C01819=1031.307,-50.754,414.134,167.850,42.108,157.823
C01820=1031.301,-51.003,414.145,167.848,42.110,157.824
C01821=1031.295,-51.252,414.157,167.845,42.111,157.824
C01822=1031.289,-51.502,414.170,167.842,42.113,157.824
C01823=1031.282,-51.752,414.182,167.840,42.114,157.824
C01824=1031.274,-52.034,414.195,167.836,42.116,157.824
C01825=1031.267,-52.314,414.209,167.834,42.117,157.824
C01826=1031.261,-52.596,414.222,167.831,42.119,157.824
C01827=1031.253,-52.877,414.236,167.827,42.120,157.824
C01828=1031.247,-53.127,414.247,167.824,42.122,157.824
C01829=1031.241,-53.376,414.259,167.822,42.123,157.824
C01830=1031.235,-53.626,414.271,167.820,42.124,157.824
C01831=1031.228,-53.875,414.283,167.817,42.126,157.824
C01832=1031.222,-54.125,414.296,167.814,42.127,157.824
C01833=1031.215,-54.375,414.308,167.811,42.128,157.824
C01834=1031.209,-54.624,414.320,167.809,42.130,157.825
C01835=1031.204,-54.874,414.331,167.806,42.131,157.825
C01836=1031.197,-55.124,414.343,167.803,42.133,157.825
C01837=1031.191,-55.373,414.355,167.800,42.134,157.825
C01838=1031.184,-55.623,414.367,167.797,42.136,157.825
C01839=1031.179,-55.872,414.379,167.795,42.137,157.825
C01840=1031.172,-56.122,414.391,167.792,42.139,157.825
C01841=1031.166,-56.372,414.402,167.789,42.140,157.825
C01842=1031.159,-56.621,414.414,167.786,42.141,157.825
C01843=1031.153,-56.871,414.427,167.783,42.143,157.825
C01844=1031.147,-57.120,414.439,167.782,42.144,157.825
C01845=1031.141,-57.370,414.450,167.779,42.145,157.825
C01846=1031.135,-57.620,414.462,167.776,42.146,157.825
C01847=1031.128,-57.870,414.474,167.773,42.148,157.826
C01848=1031.122,-58.119,414.485,167.771,42.149,157.826
C01849=1031.116,-58.369,414.497,167.768,42.150,157.826
C01850=1031.110,-58.619,414.510,167.765,42.152,157.826
C01851=1031.104,-58.867,414.521,167.762,42.153,157.826
C01852=1031.097,-59.118,414.533,167.759,42.155,157.826
C01853=1031.091,-59.367,414.545,167.757,42.156,157.826
C01854=1031.085,-59.617,414.557,167.754,42.158,157.826
C01855=1031.079,-59.867,414.568,167.751,42.159,157.826
C01856=1031.072,-60.116,414.580,167.748,42.161,157.826
C01857=1031.066,-60.366,414.592,167.745,42.162,157.826
C01858=1031.061,-60.616,414.603,167.743,42.163,157.826
C01859=1031.054,-60.865,414.615,167.740,42.165,157.826
C01860=1031.048,-61.115,414.627,167.737,42.166,157.826
C01861=1031.042,-61.364,414.638,167.735,42.168,157.826
C01862=1031.036,-61.614,414.651,167.732,42.169,157.826
C01863=1031.030,-61.864,414.662,167.730,42.170,157.827
C01864=1031.023,-62.113,414.674,167.727,42.172,157.827
C01865=1031.017,-62.363,414.685,167.724,42.173,157.827
C01866=1031.010,-62.613,414.697,167.721,42.174,157.827
C01867=1031.005,-62.862,414.709,167.718,42.176,157.827
C01868=1030.999,-63.112,414.720,167.716,42.177,157.827
C01869=1030.993,-63.361,414.732,167.713,42.178,157.827
C01870=1030.986,-63.611,414.743,167.710,42.180,157.827
C01871=1030.981,-63.861,414.756,167.707,42.181,157.827
C01872=1030.975,-64.111,414.766,167.704,42.182,157.827
C01873=1030.968,-64.360,414.778,167.702,42.184,157.827
C01874=1030.962,-64.610,414.789,167.699,42.185,157.827
C01875=1030.956,-64.859,414.801,167.696,42.187,157.827
C01876=1030.951,-65.109,414.813,167.693,42.188,157.827
C01877=1030.944,-65.359,414.825,167.690,42.189,157.827
C01878=1030.938,-65.609,414.836,167.688,42.191,157.827
C01879=1030.932,-65.858,414.848,167.685,42.192,157.828
C01880=1030.925,-66.108,414.859,167.683,42.194,157.828
C01881=1030.920,-66.357,414.871,167.680,42.195,157.828
C01882=1030.914,-66.607,414.882,167.678,42.197,157.828
C01883=1030.908,-66.857,414.893,167.675,42.198,157.828
C01884=1030.901,-67.106,414.905,167.672,42.199,157.828
C01885=1030.896,-67.356,414.916,167.669,42.201,157.828
C01886=1030.890,-67.606,414.928,167.666,42.202,157.828
C01887=1030.884,-67.855,414.939,167.664,42.204,157.828
C01888=1030.877,-68.138,414.952,167.660,42.205,157.828
C01889=1030.870,-68.421,414.965,167.657,42.207,157.828
C01890=1030.863,-68.703,414.978,167.654,42.208,157.828
C01891=1030.856,-68.986,414.991,167.651,42.210,157.828
C01892=1030.851,-69.235,415.003,167.648,42.211,157.828
C01893=1030.845,-69.485,415.014,167.646,42.212,157.828
C01894=1030.839,-69.735,415.025,167.643,42.213,157.828
C01895=1030.832,-69.984,415.037,167.640,42.215,157.829
C01896=1030.826,-70.234,415.048,167.638,42.216,157.829
C01897=1030.820,-70.484,415.059,167.635,42.217,157.829
C01898=1030.815,-70.733,415.071,167.632,42.219,157.829
C01899=1030.809,-70.983,415.083,167.629,42.220,157.829
C01900=1030.803,-71.233,415.093,167.626,42.222,157.829
C01901=1030.797,-71.481,415.105,167.624,42.223,157.829
C01902=1030.790,-71.732,415.116,167.621,42.225,157.829
C01903=1030.785,-71.981,415.127,167.618,42.226,157.829
C01904=1030.779,-72.232,415.139,167.615,42.227,157.829
C01905=1030.773,-72.481,415.151,167.612,42.229,157.829
C01906=1030.767,-72.730,415.161,167.610,42.230,157.829
C01907=1030.761,-72.980,415.173,167.607,42.232,157.829
C01908=1030.755,-73.230,415.184,167.604,42.233,157.829
C01909=1030.749,-73.480,415.195,167.601,42.234,157.829
C01910=1030.744,-73.729,415.207,167.598,42.236,157.829
C01911=1030.738,-73.979,415.218,167.596,42.237,157.829
C01912=1030.731,-74.229,415.229,167.593,42.239,157.830
C01913=1030.726,-74.478,415.240,167.590,42.240,157.830
C01914=1030.720,-74.728,415.251,167.587,42.242,157.830
C01915=1030.713,-74.978,415.262,167.584,42.243,157.830
C01916=1030.707,-75.227,415.272,167.582,42.245,157.830
C01917=1030.701,-75.477,415.284,167.579,42.246,157.830
C01918=1030.695,-75.727,415.295,167.576,42.247,157.830
C01919=1030.689,-75.976,415.305,167.574,42.249,157.830
C01920=1030.683,-76.226,415.317,167.571,42.250,157.830
C01921=1030.677,-76.475,415.328,167.568,42.252,157.830
C01922=1030.671,-76.725,415.339,167.565,42.254,157.830
C01923=1030.664,-76.975,415.350,167.562,42.255,157.830
C01924=1030.658,-77.224,415.361,167.560,42.257,157.831
C01925=1030.653,-77.474,415.372,167.557,42.258,157.831
C01926=1030.646,-77.724,415.383,167.554,42.260,157.831
C01927=1030.641,-77.973,415.394,167.551,42.261,157.831
C01928=1030.635,-78.223,415.405,167.549,42.263,157.831
C01929=1030.629,-78.474,415.415,167.546,42.264,157.831
C01930=1030.622,-78.723,415.425,167.543,42.265,157.831
C01931=1030.617,-78.972,415.436,167.540,42.267,157.831
C01932=1030.610,-79.223,415.447,167.538,42.269,157.831
C01933=1030.604,-79.472,415.458,167.534,42.270,157.831
C01934=1030.599,-79.722,415.469,167.531,42.272,157.831
C01935=1030.593,-79.971,415.480,167.528,42.273,157.831
C01936=1030.586,-80.221,415.491,167.525,42.275,157.831
C01937=1030.580,-80.470,415.502,167.523,42.277,157.832
C01938=1030.574,-80.720,415.512,167.520,42.279,157.832
C01939=1030.568,-80.970,415.522,167.517,42.280,157.832
C01940=1030.562,-81.220,415.533,167.515,42.281,157.832
C01941=1030.555,-81.469,415.544,167.512,42.283,157.832
C01942=1030.549,-81.719,415.555,167.509,42.285,157.832
C01943=1030.543,-81.969,415.566,167.506,42.287,157.832
C01944=1030.537,-82.219,415.575,167.503,42.288,157.832
C01945=1030.531,-82.468,415.586,167.500,42.290,157.832
C01946=1030.524,-82.718,415.597,167.497,42.292,157.832
C01947=1030.519,-82.967,415.608,167.495,42.293,157.833
C01948=1030.513,-83.218,415.618,167.492,42.295,157.833
C01949=1030.507,-83.467,415.628,167.489,42.296,157.833
C01950=1030.500,-83.717,415.639,167.486,42.298,157.833
C01951=1030.494,-83.967,415.649,167.484,42.300,157.833
C01952=1030.487,-84.251,415.662,167.480,42.302,157.833
C01953=1030.480,-84.535,415.674,167.477,42.304,157.833
C01954=1030.474,-84.820,415.685,167.474,42.306,157.833
C01955=1030.467,-85.105,415.697,167.471,42.307,157.833
C01956=1030.461,-85.354,415.708,167.468,42.309,157.834
C01957=1030.455,-85.604,415.718,167.464,42.310,157.834
C01958=1030.449,-85.854,415.729,167.462,42.312,157.834
C01959=1030.443,-86.104,415.739,167.459,42.314,157.834
C01960=1030.437,-86.353,415.750,167.456,42.316,157.834
C01961=1030.430,-86.603,415.760,167.453,42.317,157.834
C01962=1030.425,-86.853,415.770,167.451,42.319,157.834
C01963=1030.418,-87.102,415.780,167.448,42.321,157.834
C01964=1030.412,-87.352,415.791,167.445,42.322,157.834
C01965=1030.407,-87.602,415.802,167.442,42.323,157.834
C01966=1030.400,-87.851,415.812,167.439,42.325,157.834
C01967=1030.395,-88.101,415.822,167.436,42.327,157.835
C01968=1030.388,-88.351,415.832,167.433,42.329,157.835
C01969=1030.383,-88.601,415.843,167.431,42.331,157.835
C01970=1030.376,-88.850,415.853,167.428,42.332,157.835
C01971=1030.371,-89.100,415.863,167.425,42.334,157.835
C01972=1030.364,-89.349,415.873,167.422,42.336,157.835
C01973=1030.358,-89.599,415.885,167.420,42.337,157.835
C01974=1030.353,-89.849,415.895,167.417,42.338,157.835
C01975=1030.346,-90.099,415.905,167.413,42.340,157.835
C01976=1030.341,-90.349,415.915,167.410,42.342,157.835
C01977=1030.334,-90.598,415.925,167.408,42.344,157.836
C01978=1030.329,-90.848,415.936,167.405,42.346,157.836
C01979=1030.323,-91.098,415.945,167.402,42.347,157.836
C01980=1030.317,-91.347,415.956,167.399,42.349,157.836
C01981=1030.311,-91.597,415.966,167.397,42.350,157.836
C01982=1030.305,-91.847,415.976,167.394,42.352,157.836
C01983=1030.299,-92.096,415.986,167.391,42.353,157.836
C01984=1030.293,-92.346,415.997,167.388,42.355,157.836
C01985=1030.287,-92.596,416.006,167.385,42.357,157.836
C01986=1030.282,-92.846,416.017,167.382,42.359,157.836
C01987=1030.275,-93.095,416.027,167.379,42.360,157.836
C01988=1030.270,-93.345,416.037,167.377,42.362,157.836
C01989=1030.264,-93.595,416.048,167.374,42.364,157.837
C01990=1030.258,-93.844,416.058,167.371,42.365,157.837
C01991=1030.252,-94.095,416.068,167.369,42.367,157.837
C01992=1030.246,-94.344,416.078,167.366,42.368,157.837
C01993=1030.240,-94.594,416.088,167.362,42.370,157.837
C01994=1030.234,-94.844,416.098,167.359,42.372,157.837
C01995=1030.228,-95.093,416.109,167.357,42.374,157.837
C01996=1030.222,-95.343,416.118,167.354,42.375,157.837
C01997=1030.217,-95.593,416.128,167.351,42.377,157.837
C01998=1030.210,-95.842,416.139,167.348,42.379,157.837
C01999=1030.205,-96.092,416.149,167.346,42.380,157.838
C02000=1030.199,-96.342,416.158,167.343,42.382,157.838
C02001=1030.193,-96.592,416.169,167.340,42.383,157.838
C02002=1030.187,-96.841,416.179,167.336,42.385,157.838
C02003=1030.182,-97.091,416.189,167.334,42.387,157.838
C02004=1030.176,-97.341,416.198,167.331,42.389,157.838
C02005=1030.170,-97.590,416.209,167.328,42.390,157.838
C02006=1030.164,-97.840,416.219,167.325,42.392,157.838
C02007=1030.158,-98.090,416.228,167.323,42.394,157.838
C02008=1030.152,-98.339,416.238,167.320,42.395,157.838
C02009=1030.146,-98.590,416.248,167.316,42.397,157.839
C02010=1030.140,-98.839,416.257,167.314,42.399,157.839
C02011=1030.134,-99.089,416.267,167.311,42.401,157.839
C02012=1030.127,-99.338,416.277,167.308,42.403,157.839
C02013=1030.122,-99.588,416.287,167.306,42.405,157.839
C02014=1030.116,-99.838,416.297,167.302,42.407,157.839
C02015=1030.110,-100.087,416.306,167.299,42.408,157.839
C02016=1030.103,-100.375,416.317,167.297,42.410,157.839
C02017=1030.096,-100.661,416.328,167.293,42.413,157.840
C02018=1030.090,-100.948,416.340,167.289,42.415,157.840
C02019=1030.083,-101.236,416.351,167.287,42.417,157.840
C02020=1030.077,-101.485,416.360,167.284,42.418,157.840
C02021=1030.071,-101.734,416.370,167.280,42.420,157.840
C02022=1030.065,-101.984,416.379,167.278,42.422,157.840
C02023=1030.060,-102.234,416.389,167.275,42.424,157.840
C02024=1030.053,-102.484,416.399,167.272,42.426,157.840
C02025=1030.047,-102.734,416.409,167.269,42.428,157.840
C02026=1030.042,-102.983,416.418,167.266,42.429,157.841
C02027=1030.035,-103.233,416.427,167.263,42.431,157.841
C02028=1030.030,-103.483,416.438,167.260,42.433,157.841
C02029=1030.024,-103.733,416.447,167.258,42.435,157.841
C02030=1030.018,-103.983,416.457,167.255,42.437,157.841
C02031=1030.012,-104.232,416.466,167.252,42.439,157.841
C02032=1030.006,-104.481,416.475,167.249,42.440,157.841
C02033=1030.001,-104.732,416.486,167.246,42.442,157.841
C02034=1029.994,-104.981,416.495,167.243,42.444,157.842
C02035=1029.988,-105.231,416.505,167.241,42.446,157.842
C02036=1029.983,-105.480,416.514,167.238,42.448,157.842
C02037=1029.976,-105.730,416.524,167.234,42.450,157.842
C02038=1029.970,-105.980,416.533,167.231,42.451,157.842
C02039=1029.965,-106.230,416.543,167.229,42.453,157.842
C02040=1029.960,-106.480,416.552,167.226,42.455,157.842
C02041=1029.953,-106.729,416.561,167.223,42.457,157.842
C02042=1029.947,-106.979,416.571,167.220,42.459,157.842
C02043=1029.941,-107.229,416.580,167.217,42.461,157.843
C02044=1029.935,-107.478,416.590,167.214,42.462,157.843
C02045=1029.930,-107.729,416.598,167.212,42.464,157.843
C02046=1029.923,-107.978,416.608,167.209,42.466,157.843
C02047=1029.918,-108.227,416.617,167.205,42.468,157.843
C02048=1029.912,-108.477,416.627,167.203,42.470,157.843
C02049=1029.906,-108.727,416.636,167.200,42.472,157.843
C02050=1029.900,-108.977,416.645,167.197,42.473,157.843
C02051=1029.894,-109.227,416.654,167.195,42.475,157.843
C02052=1029.888,-109.476,416.664,167.191,42.478,157.844
C02053=1029.882,-109.727,416.673,167.188,42.480,157.844
C02054=1029.876,-109.976,416.682,167.186,42.482,157.844
C02055=1029.870,-110.226,416.692,167.183,42.483,157.844
C02056=1029.864,-110.475,416.701,167.179,42.485,157.844
C02057=1029.859,-110.725,416.710,167.177,42.487,157.844
C02058=1029.853,-110.975,416.719,167.174,42.489,157.844
C02059=1029.847,-111.225,416.729,167.171,42.491,157.845
C02060=1029.841,-111.474,416.737,167.168,42.493,157.845
C02061=1029.835,-111.724,416.747,167.165,42.495,157.845
C02062=1029.829,-111.975,416.756,167.162,42.497,157.845
C02063=1029.824,-112.224,416.765,167.160,42.499,157.845
C02064=1029.817,-112.474,416.774,167.157,42.501,157.845
C02065=1029.812,-112.723,416.783,167.153,42.503,157.845
C02066=1029.806,-112.973,416.793,167.151,42.504,157.845
C02067=1029.800,-113.223,416.802,167.148,42.506,157.846
C02068=1029.795,-113.473,416.811,167.145,42.508,157.846
C02069=1029.788,-113.722,416.820,167.143,42.511,157.846
C02070=1029.783,-113.972,416.829,167.139,42.513,157.846
C02071=1029.777,-114.222,416.838,167.136,42.514,157.846
C02072=1029.771,-114.472,416.847,167.134,42.516,157.846
C02073=1029.766,-114.721,416.856,167.131,42.518,157.846
C02074=1029.760,-114.972,416.865,167.127,42.520,157.846
C02075=1029.754,-115.221,416.874,167.125,42.522,157.847
C02076=1029.748,-115.471,416.883,167.122,42.524,157.847
C02077=1029.742,-115.720,416.892,167.119,42.526,157.847
C02078=1029.736,-115.971,416.901,167.116,42.528,157.847
C02079=1029.731,-116.220,416.910,167.113,42.530,157.847
C02080=1029.724,-116.506,416.921,167.109,42.533,157.847
C02081=1029.717,-116.793,416.930,167.107,42.534,157.847
C02082=1029.711,-117.079,416.941,167.103,42.537,157.848
C02083=1029.703,-117.365,416.951,167.100,42.539,157.848
C02084=1029.698,-117.615,416.960,167.097,42.541,157.848
C02085=1029.692,-117.866,416.968,167.094,42.543,157.848
C02086=1029.686,-118.115,416.978,167.091,42.545,157.848
C02087=1029.680,-118.365,416.986,167.088,42.547,157.848
C02088=1029.674,-118.614,416.995,167.085,42.550,157.849
C02089=1029.668,-118.864,417.004,167.083,42.551,157.849
C02090=1029.663,-119.114,417.012,167.079,42.553,157.849
C02091=1029.657,-119.364,417.022,167.076,42.555,157.849
C02092=1029.651,-119.613,417.030,167.074,42.558,157.849
C02093=1029.645,-119.864,417.039,167.071,42.560,157.849
C02094=1029.639,-120.113,417.048,167.067,42.562,157.849
C02095=1029.634,-120.362,417.056,167.065,42.563,157.849
C02096=1029.628,-120.612,417.065,167.062,42.566,157.850
C02097=1029.622,-120.862,417.073,167.060,42.568,157.850
C02098=1029.616,-121.112,417.083,167.056,42.570,157.850
C02099=1029.611,-121.362,417.091,167.053,42.571,157.850
C02100=1029.605,-121.612,417.100,167.051,42.574,157.850
C02101=1029.599,-121.861,417.109,167.048,42.576,157.850
C02102=1029.593,-122.111,417.117,167.044,42.578,157.850
C02103=1029.588,-122.361,417.126,167.042,42.580,157.851
C02104=1029.582,-122.610,417.134,167.039,42.582,157.851
C02105=1029.576,-122.861,417.143,167.036,42.584,157.851
C02106=1029.570,-123.110,417.152,167.033,42.586,157.851
C02107=1029.564,-123.360,417.161,167.030,42.588,157.851
C02108=1029.558,-123.610,417.169,167.028,42.590,157.851
C02109=1029.553,-123.859,417.177,167.025,42.592,157.851
C02110=1029.547,-124.110,417.186,167.021,42.594,157.852
C02111=1029.542,-124.359,417.195,167.019,42.597,157.852
C02112=1029.536,-124.608,417.203,167.016,42.598,157.852
C02113=1029.530,-124.859,417.212,167.012,42.600,157.852
C02114=1029.524,-125.108,417.220,167.010,42.603,157.852
C02115=1029.518,-125.359,417.229,167.007,42.605,157.852
C02116=1029.513,-125.608,417.237,167.004,42.607,157.852
C02117=1029.507,-125.858,417.245,167.001,42.609,157.853
C02118=1029.501,-126.108,417.254,166.998,42.611,157.853
C02119=1029.495,-126.358,417.262,166.996,42.614,157.853
C02120=1029.489,-126.607,417.270,166.992,42.615,157.853
C02121=1029.484,-126.858,417.279,166.989,42.617,157.853
C02122=1029.478,-127.107,417.287,166.987,42.620,157.853
C02123=1029.472,-127.357,417.295,166.984,42.622,157.854
C02124=1029.466,-127.606,417.304,166.980,42.624,157.854
C02125=1029.461,-127.855,417.313,166.978,42.626,157.854
C02126=1029.455,-128.106,417.321,166.975,42.628,157.854
C02127=1029.450,-128.355,417.331,166.972,42.629,157.854
C02128=1029.446,-128.604,417.340,166.970,42.630,157.854
C02129=1029.443,-128.855,417.351,166.968,42.631,157.854
C02130=1029.440,-129.104,417.362,166.964,42.630,157.854
C02131=1029.437,-129.354,417.374,166.962,42.630,157.853
C02132=1029.436,-129.604,417.386,166.960,42.629,157.853
C02133=1029.435,-129.853,417.399,166.958,42.627,157.853
C02134=1029.435,-130.103,417.412,166.955,42.625,157.852
C02135=1029.435,-130.353,417.426,166.954,42.623,157.852
C02136=1029.435,-130.603,417.440,166.952,42.620,157.851
C02137=1029.436,-130.853,417.456,166.950,42.617,157.850
C02138=1029.439,-131.103,417.472,166.948,42.613,157.850
C02139=1029.441,-131.352,417.488,166.947,42.608,157.849
C02140=1029.445,-131.603,417.505,166.945,42.604,157.848
C02141=1029.448,-131.853,417.523,166.944,42.599,157.847
C02142=1029.453,-132.103,417.540,166.942,42.593,157.846
C02143=1029.458,-132.352,417.560,166.941,42.586,157.845
C02144=1029.141,-132.377,417.253,166.892,42.832,157.882
C02145=1029.137,-132.128,417.233,166.894,42.838,157.883
C02146=1029.132,-131.879,417.215,166.895,42.844,157.884
C02147=1029.128,-131.628,417.198,166.896,42.849,157.885
C02148=1029.125,-131.378,417.181,166.898,42.854,157.886
C02149=1029.122,-131.128,417.165,166.900,42.858,157.887
C02150=1029.120,-130.878,417.149,166.902,42.862,157.888
C02151=1029.119,-130.628,417.133,166.903,42.865,157.889
C02152=1029.118,-130.378,417.119,166.905,42.868,157.889
C02153=1029.118,-130.128,417.105,166.907,42.871,157.890
C02154=1029.118,-129.878,417.092,166.909,42.872,157.890
C02155=1029.119,-129.629,417.078,166.911,42.874,157.891
C02156=1029.121,-129.379,417.066,166.914,42.875,157.891
C02157=1029.123,-129.129,417.054,166.916,42.876,157.891
C02158=1029.126,-128.880,417.044,166.918,42.876,157.891
C02159=1029.129,-128.630,417.033,166.921,42.876,157.892
C02160=1029.134,-128.381,417.023,166.923,42.875,157.892
C02161=1029.138,-128.131,417.014,166.926,42.873,157.892
C02162=1029.143,-127.880,417.005,166.929,42.872,157.891
C02163=1029.150,-127.631,416.996,166.932,42.869,157.891
C02164=1029.155,-127.382,416.988,166.935,42.867,157.891
C02165=1029.161,-127.132,416.980,166.937,42.865,157.891
C02166=1029.166,-126.882,416.971,166.941,42.863,157.891
C02167=1029.173,-126.632,416.963,166.944,42.861,157.891
C02168=1029.178,-126.383,416.955,166.946,42.858,157.891
C02169=1029.184,-126.133,416.947,166.950,42.856,157.890
C02170=1029.190,-125.883,416.938,166.953,42.854,157.890
C02171=1029.195,-125.633,416.929,166.955,42.852,157.890
C02172=1029.201,-125.384,416.921,166.959,42.850,157.890
C02173=1029.207,-125.133,416.913,166.961,42.847,157.890
C02174=1029.213,-124.884,416.905,166.964,42.845,157.890
C02175=1029.218,-124.634,416.896,166.968,42.843,157.889
C02176=1029.224,-124.384,416.887,166.970,42.841,157.889
C02177=1029.230,-124.135,416.879,166.973,42.839,157.889
C02178=1029.236,-123.885,416.870,166.975,42.836,157.889
C02179=1029.242,-123.635,416.861,166.979,42.834,157.889
C02180=1029.247,-123.385,416.853,166.982,42.833,157.889
C02181=1029.253,-123.136,416.845,166.984,42.830,157.889
C02182=1029.259,-122.886,416.835,166.988,42.828,157.888
C02183=1029.264,-122.636,416.827,166.991,42.826,157.888
C02184=1029.271,-122.386,416.819,166.993,42.824,157.888
C02185=1029.276,-122.136,416.810,166.996,42.822,157.888
C02186=1029.281,-121.887,416.802,166.999,42.820,157.888
C02187=1029.288,-121.637,416.792,167.002,42.817,157.888
C02188=1029.294,-121.387,416.784,167.005,42.816,157.888
C02189=1029.299,-121.137,416.775,167.008,42.814,157.888
C02190=1029.305,-120.887,416.767,167.011,42.811,157.887
C02191=1029.311,-120.638,416.757,167.013,42.809,157.887
C02192=1029.317,-120.388,416.750,167.016,42.807,157.887
C02193=1029.322,-120.138,416.741,167.020,42.805,157.887
C02194=1029.328,-119.889,416.731,167.022,42.803,157.887
C02195=1029.334,-119.639,416.723,167.025,42.801,157.887
C02196=1029.339,-119.388,416.714,167.029,42.799,157.887
C02197=1029.345,-119.139,416.706,167.031,42.796,157.886
C02198=1029.352,-118.889,416.697,167.034,42.795,157.886
C02199=1029.357,-118.640,416.688,167.037,42.793,157.886
C02200=1029.363,-118.390,416.679,167.040,42.791,157.886
C02201=1029.369,-118.140,416.671,167.043,42.788,157.886
C02202=1029.375,-117.890,416.662,167.045,42.786,157.886
C02203=1029.380,-117.641,416.653,167.049,42.784,157.886
C02204=1029.386,-117.390,416.644,167.052,42.782,157.885
C02205=1029.393,-117.105,416.634,167.055,42.780,157.885
C02206=1029.400,-116.818,416.624,167.058,42.777,157.885
C02207=1029.406,-116.532,416.614,167.061,42.775,157.885
C02208=1029.413,-116.245,416.603,167.065,42.773,157.885
C02209=1029.418,-115.996,416.595,167.068,42.771,157.885
C02210=1029.425,-115.746,416.585,167.070,42.769,157.885
C02211=1029.430,-115.496,416.576,167.074,42.766,157.884
C02212=1029.437,-115.247,416.567,167.077,42.764,157.884
C02213=1029.442,-114.997,416.559,167.079,42.763,157.884
C02214=1029.448,-114.747,416.549,167.082,42.761,157.884
C02215=1029.454,-114.497,416.541,167.085,42.758,157.884
C02216=1029.460,-114.248,416.531,167.088,42.756,157.884
C02217=1029.465,-113.997,416.523,167.091,42.754,157.884
C02218=1029.471,-113.748,416.513,167.093,42.753,157.883
C02219=1029.477,-113.498,416.504,167.097,42.751,157.883
C02220=1029.482,-113.249,416.495,167.100,42.748,157.883
C02221=1029.488,-112.998,416.486,167.102,42.746,157.883
C02222=1029.495,-112.748,416.477,167.105,42.744,157.883
C02223=1029.500,-112.499,416.468,167.109,42.742,157.883
C02224=1029.506,-112.249,416.459,167.111,42.741,157.883
C02225=1029.512,-112.000,416.450,167.114,42.739,157.883
C02226=1029.517,-111.749,416.441,167.117,42.737,157.882
C02227=1029.524,-111.500,416.431,167.120,42.734,157.882
C02228=1029.529,-111.251,416.422,167.123,42.732,157.882
C02229=1029.535,-111.000,416.413,167.126,42.731,157.882
C02230=1029.541,-110.750,416.404,167.128,42.729,157.882
C02231=1029.547,-110.501,416.394,167.132,42.727,157.882
C02232=1029.553,-110.251,416.386,167.135,42.725,157.882
C02233=1029.559,-110.001,416.376,167.137,42.722,157.881
C02234=1029.564,-109.752,416.367,167.140,42.721,157.881
C02235=1029.570,-109.501,416.358,167.143,42.719,157.881
C02236=1029.576,-109.252,416.348,167.146,42.717,157.881
C02237=1029.582,-109.003,416.339,167.149,42.715,157.881
C02238=1029.588,-108.753,416.330,167.151,42.713,157.881
C02239=1029.594,-108.502,416.321,167.155,42.711,157.881
C02240=1029.600,-108.253,416.312,167.158,42.709,157.881
C02241=1029.606,-108.003,416.302,167.160,42.707,157.880
C02242=1029.612,-107.754,416.292,167.163,42.705,157.880
C02243=1029.618,-107.503,416.284,167.167,42.703,157.880
C02244=1029.623,-107.254,416.274,167.169,42.701,157.880
C02245=1029.630,-107.004,416.265,167.172,42.699,157.880
C02246=1029.636,-106.755,416.255,167.175,42.698,157.880
C02247=1029.641,-106.505,416.246,167.178,42.696,157.880
C02248=1029.647,-106.255,416.237,167.181,42.693,157.880
C02249=1029.653,-106.005,416.228,167.184,42.691,157.879
C02250=1029.659,-105.755,416.217,167.186,42.689,157.879
C02251=1029.664,-105.506,416.208,167.189,42.688,157.879
C02252=1029.670,-105.256,416.199,167.193,42.686,157.879
C02253=1029.677,-105.006,416.189,167.195,42.684,157.879
C02254=1029.683,-104.757,416.180,167.198,42.682,157.879
C02255=1029.688,-104.508,416.170,167.201,42.680,157.879
C02256=1029.694,-104.257,416.161,167.204,42.678,157.879
C02257=1029.700,-104.007,416.151,167.207,42.676,157.879
C02258=1029.706,-103.757,416.142,167.210,42.674,157.878
C02259=1029.711,-103.508,416.133,167.212,42.673,157.878
C02260=1029.718,-103.258,416.123,167.215,42.671,157.878
C02261=1029.723,-103.008,416.113,167.219,42.669,157.878
C02262=1029.729,-102.758,416.103,167.222,42.667,157.878
C02263=1029.735,-102.509,416.094,167.224,42.665,157.878
C02264=1029.741,-102.260,416.084,167.227,42.663,157.878
C02265=1029.746,-102.009,416.074,167.230,42.662,157.878
C02266=1029.753,-101.760,416.065,167.233,42.660,157.878
C02267=1029.759,-101.510,416.055,167.236,42.658,157.877
C02268=1029.765,-101.260,416.046,167.239,42.656,157.877
C02269=1029.772,-100.973,416.035,167.242,42.653,157.877
C02270=1029.778,-100.687,416.024,167.245,42.651,157.877
C02271=1029.785,-100.400,416.011,167.248,42.649,157.877
C02272=1029.792,-100.113,416.000,167.252,42.647,157.877
C02273=1029.798,-99.863,415.991,167.255,42.646,157.877
C02274=1029.804,-99.614,415.981,167.257,42.643,157.876
C02275=1029.810,-99.365,415.972,167.260,42.641,157.876
C02276=1029.815,-99.114,415.962,167.264,42.639,157.876
C02277=1029.821,-98.865,415.952,167.266,42.638,157.876
C02278=1029.828,-98.615,415.943,167.269,42.636,157.876
C02279=1029.834,-98.365,415.933,167.272,42.634,157.876
C02280=1029.839,-98.116,415.922,167.274,42.632,157.876
C02281=1029.846,-97.866,415.913,167.278,42.630,157.876
C02282=1029.852,-97.616,415.903,167.281,42.628,157.876
C02283=1029.857,-97.366,415.893,167.284,42.627,157.876
C02284=1029.863,-97.116,415.884,167.286,42.625,157.875
C02285=1029.869,-96.866,415.873,167.289,42.623,157.875
C02286=1029.875,-96.617,415.863,167.292,42.622,157.875
C02287=1029.880,-96.367,415.853,167.295,42.620,157.875
C02288=1029.886,-96.118,415.844,167.298,42.618,157.875
C02289=1029.892,-95.868,415.833,167.301,42.617,157.875
C02290=1029.898,-95.618,415.823,167.304,42.615,157.875
C02291=1029.904,-95.368,415.813,167.306,42.613,157.875
C02292=1029.910,-95.118,415.804,167.309,42.611,157.875
C02293=1029.916,-94.869,415.793,167.312,42.609,157.875
C02294=1029.922,-94.619,415.783,167.315,42.607,157.874
C02295=1029.927,-94.369,415.773,167.318,42.606,157.874
C02296=1029.934,-94.120,415.763,167.321,42.605,157.874
C02297=1029.939,-93.870,415.752,167.324,42.603,157.874
C02298=1029.945,-93.620,415.743,167.326,42.601,157.874
C02299=1029.951,-93.370,415.732,167.329,42.599,157.874
C02300=1029.957,-93.121,415.722,167.332,42.597,157.874
C02301=1029.963,-92.871,415.712,167.336,42.596,157.874
C02302=1029.969,-92.621,415.702,167.338,42.594,157.874
C02303=1029.975,-92.371,415.692,167.341,42.592,157.874
C02304=1029.981,-92.122,415.682,167.344,42.591,157.873
C02305=1029.986,-91.872,415.671,167.346,42.589,157.873
C02306=1029.993,-91.623,415.661,167.349,42.587,157.873
C02307=1029.998,-91.373,415.651,167.352,42.586,157.873
C02308=1030.005,-91.123,415.641,167.354,42.584,157.873
C02309=1030.010,-90.873,415.631,167.358,42.582,157.873
C02310=1030.016,-90.623,415.620,167.361,42.580,157.873
C02311=1030.022,-90.374,415.610,167.364,42.578,157.873
C02312=1030.028,-90.124,415.600,167.366,42.577,157.873
C02313=1030.034,-89.875,415.590,167.369,42.575,157.873
C02314=1030.040,-89.625,415.579,167.372,42.574,157.873
C02315=1030.046,-89.375,415.569,167.374,42.572,157.872
C02316=1030.051,-89.125,415.559,167.378,42.570,157.872
C02317=1030.058,-88.876,415.549,167.381,42.568,157.872
C02318=1030.064,-88.625,415.538,167.384,42.566,157.872
C02319=1030.070,-88.376,415.528,167.386,42.565,157.872
C02320=1030.076,-88.127,415.517,167.389,42.563,157.872
C02321=1030.082,-87.877,415.507,167.392,42.561,157.872
C02322=1030.088,-87.627,415.497,167.394,42.560,157.872
C02323=1030.094,-87.377,415.486,167.398,42.558,157.872
C02324=1030.100,-87.128,415.476,167.401,42.556,157.872
C02325=1030.105,-86.878,415.466,167.404,42.555,157.872
C02326=1030.113,-86.628,415.455,167.406,42.553,157.871
C02327=1030.118,-86.379,415.444,167.409,42.551,157.871
C02328=1030.124,-86.129,415.434,167.412,42.549,157.871
C02329=1030.130,-85.879,415.424,167.414,42.547,157.871
C02330=1030.136,-85.629,415.414,167.418,42.545,157.871
C02331=1030.142,-85.380,415.404,167.421,42.544,157.871
C02332=1030.148,-85.130,415.392,167.424,42.543,157.871
C02333=1030.155,-84.845,415.380,167.426,42.541,157.871
C02334=1030.163,-84.561,415.369,167.430,42.539,157.871
C02335=1030.169,-84.276,415.357,167.433,42.537,157.870
C02336=1030.176,-83.992,415.345,167.436,42.534,157.870
C02337=1030.182,-83.742,415.334,167.439,42.533,157.870
C02338=1030.188,-83.493,415.324,167.442,42.531,157.870
C02339=1030.194,-83.243,415.314,167.444,42.530,157.870
C02340=1030.201,-82.993,415.303,167.448,42.528,157.870
C02341=1030.207,-82.743,415.292,167.451,42.526,157.870
C02342=1030.212,-82.493,415.282,167.454,42.524,157.870
C02343=1030.218,-82.244,415.272,167.456,42.523,157.870
C02344=1030.225,-81.994,415.261,167.459,42.521,157.870
C02345=1030.231,-81.745,415.250,167.462,42.519,157.869
C02346=1030.237,-81.495,415.240,167.464,42.517,157.869
C02347=1030.242,-81.245,415.229,167.468,42.515,157.869
C02348=1030.250,-80.995,415.219,167.471,42.514,157.869
C02349=1030.255,-80.746,415.208,167.474,42.513,157.869
C02350=1030.261,-80.496,415.197,167.476,42.511,157.869
C02351=1030.268,-80.246,415.187,167.479,42.509,157.869
C02352=1030.274,-79.996,415.176,167.482,42.507,157.869
C02353=1030.279,-79.747,415.165,167.484,42.505,157.869
C02354=1030.286,-79.498,415.155,167.487,42.504,157.869
C02355=1030.292,-79.247,415.144,167.490,42.502,157.868
C02356=1030.298,-78.998,415.133,167.493,42.501,157.868
C02357=1030.304,-78.749,415.122,167.495,42.499,157.868
C02358=1030.310,-78.498,415.111,167.499,42.497,157.868
C02359=1030.316,-78.249,415.100,167.502,42.496,157.868
C02360=1030.321,-77.999,415.089,167.505,42.495,157.868
C02361=1030.328,-77.749,415.078,167.507,42.493,157.868
C02362=1030.334,-77.499,415.068,167.510,42.491,157.868
C02363=1030.340,-77.250,415.057,167.513,42.490,157.868
C02364=1030.345,-77.000,415.046,167.516,42.488,157.868
C02365=1030.352,-76.750,415.035,167.518,42.486,157.868
C02366=1030.357,-76.501,415.024,167.521,42.485,157.868
C02367=1030.364,-76.250,415.013,167.524,42.483,157.867
C02368=1030.370,-76.002,415.001,167.527,42.481,157.867
C02369=1030.376,-75.752,414.991,167.529,42.480,157.867
C02370=1030.383,-75.502,414.980,167.532,42.479,157.867
C02371=1030.388,-75.253,414.969,167.535,42.477,157.867
C02372=1030.394,-75.003,414.958,167.538,42.476,157.867
C02373=1030.400,-74.753,414.947,167.541,42.474,157.867
C02374=1030.406,-74.504,414.936,167.544,42.473,157.867
C02375=1030.412,-74.254,414.925,167.547,42.471,157.867
C02376=1030.418,-74.004,414.914,167.550,42.469,157.867
C02377=1030.424,-73.754,414.903,167.552,42.468,157.867
C02378=1030.430,-73.504,414.892,167.555,42.466,157.867
C02379=1030.436,-73.255,414.880,167.558,42.465,157.867
C02380=1030.442,-73.006,414.869,167.561,42.463,157.866
C02381=1030.448,-72.755,414.858,167.564,42.462,157.866
C02382=1030.453,-72.506,414.847,167.566,42.460,157.866
C02383=1030.459,-72.256,414.836,167.569,42.459,157.866
C02384=1030.466,-72.007,414.824,167.572,42.458,157.866
C02385=1030.472,-71.757,414.813,167.575,42.456,157.866
C02386=1030.478,-71.507,414.802,167.578,42.455,157.866
C02387=1030.484,-71.258,414.791,167.580,42.453,157.866
C02388=1030.489,-71.008,414.779,167.583,42.452,157.866
C02389=1030.495,-70.758,414.767,167.586,42.450,157.866
C02390=1030.501,-70.509,414.756,167.589,42.449,157.866
C02391=1030.508,-70.259,414.745,167.591,42.447,157.866
C02392=1030.513,-70.010,414.734,167.594,42.446,157.866
C02393=1030.519,-69.759,414.722,167.597,42.444,157.866
C02394=1030.525,-69.510,414.711,167.600,42.443,157.866
C02395=1030.531,-69.260,414.699,167.602,42.441,157.866
C02396=1030.537,-69.011,414.688,167.604,42.440,157.866
C02397=1030.544,-68.728,414.675,167.608,42.439,157.865
C02398=1030.551,-68.445,414.662,167.611,42.437,157.865
C02399=1030.557,-68.164,414.649,167.614,42.435,157.865
C02400=1030.565,-67.882,414.636,167.617,42.434,157.865
C02401=1030.570,-67.631,414.625,167.620,42.433,157.865
C02402=1030.576,-67.382,414.614,167.623,42.431,157.865
C02403=1030.583,-67.132,414.602,167.626,42.430,157.865
C02404=1030.588,-66.883,414.591,167.628,42.428,157.865
C02405=1030.595,-66.633,414.579,167.631,42.427,157.865
C02406=1030.600,-66.383,414.567,167.634,42.425,157.865
C02407=1030.607,-66.134,414.555,167.637,42.424,157.865
C02408=1030.612,-65.884,414.545,167.639,42.422,157.865
C02409=1030.619,-65.634,414.533,167.642,42.421,157.865
C02410=1030.625,-65.385,414.522,167.645,42.419,157.865
C02411=1030.630,-65.135,414.510,167.648,42.418,157.865
C02412=1030.637,-64.885,414.498,167.650,42.416,157.864
C02413=1030.643,-64.636,414.487,167.653,42.415,157.864
C02414=1030.649,-64.386,414.475,167.656,42.413,157.864
C02415=1030.655,-64.136,414.464,167.659,42.412,157.864
C02416=1030.661,-63.887,414.452,167.662,42.410,157.864
C02417=1030.667,-63.637,414.441,167.664,42.409,157.864
C02418=1030.673,-63.387,414.429,167.667,42.407,157.864
C02419=1030.680,-63.137,414.418,167.670,42.406,157.864
C02420=1030.685,-62.888,414.405,167.673,42.405,157.864
C02421=1030.691,-62.638,414.394,167.676,42.403,157.864
C02422=1030.698,-62.388,414.382,167.678,42.402,157.864
C02423=1030.704,-62.139,414.371,167.681,42.400,157.864
C02424=1030.710,-61.889,414.359,167.684,42.399,157.864
C02425=1030.716,-61.640,414.347,167.687,42.398,157.864
C02426=1030.722,-61.390,414.336,167.688,42.396,157.863
C02427=1030.729,-61.140,414.324,167.691,42.395,157.863
C02428=1030.734,-60.891,414.313,167.694,42.393,157.863
C02429=1030.740,-60.641,414.301,167.697,42.392,157.863
C02430=1030.747,-60.391,414.289,167.699,42.390,157.863
C02431=1030.753,-60.142,414.278,167.702,42.389,157.863
C02432=1030.759,-59.892,414.266,167.705,42.387,157.863
C02433=1030.765,-59.642,414.253,167.708,42.386,157.863
C02434=1030.771,-59.393,414.242,167.711,42.384,157.863
C02435=1030.778,-59.143,414.230,167.713,42.383,157.863
C02436=1030.784,-58.894,414.218,167.716,42.381,157.863
C02437=1030.790,-58.643,414.207,167.719,42.380,157.863
C02438=1030.796,-58.394,414.195,167.722,42.378,157.863
C02439=1030.803,-58.145,414.183,167.724,42.377,157.863
C02440=1030.809,-57.895,414.172,167.727,42.376,157.862
C02441=1030.814,-57.646,414.160,167.730,42.374,157.862
C02442=1030.821,-57.396,414.148,167.733,42.373,157.862
C02443=1030.828,-57.146,414.136,167.736,42.372,157.862
C02444=1030.834,-56.896,414.124,167.738,42.370,157.862
C02445=1030.839,-56.647,414.112,167.741,42.369,157.862
C02446=1030.846,-56.397,414.100,167.744,42.367,157.862
C02447=1030.853,-56.148,414.088,167.747,42.366,157.862
C02448=1030.859,-55.898,414.077,167.749,42.364,157.862
C02449=1030.864,-55.648,414.065,167.752,42.363,157.862
C02450=1030.871,-55.399,414.053,167.755,42.361,157.862
C02451=1030.877,-55.149,414.041,167.758,42.360,157.862
C02452=1030.883,-54.899,414.029,167.760,42.358,157.862
C02453=1030.890,-54.649,414.017,167.763,42.357,157.862
C02454=1030.896,-54.400,414.006,167.766,42.355,157.861
C02455=1030.902,-54.151,413.994,167.769,42.354,157.861
C02456=1030.908,-53.901,413.981,167.771,42.352,157.861
C02457=1030.915,-53.651,413.969,167.773,42.351,157.861
C02458=1030.921,-53.401,413.958,167.776,42.350,157.861
C02459=1030.927,-53.151,413.945,167.779,42.348,157.861
C02460=1030.933,-52.902,413.934,167.782,42.347,157.861
C02461=1030.941,-52.621,413.920,167.785,42.345,157.861
C02462=1030.948,-52.340,413.906,167.788,42.344,157.861
C02463=1030.955,-52.059,413.892,167.791,42.342,157.861
C02464=1030.962,-51.778,413.879,167.795,42.340,157.861
C02465=1030.969,-51.528,413.867,167.797,42.339,157.861
C02466=1030.974,-51.279,413.855,167.800,42.337,157.861
C02467=1030.981,-51.029,413.843,167.802,42.335,157.860
C02468=1030.988,-50.780,413.831,167.805,42.334,157.860
C02469=1030.994,-50.530,413.819,167.808,42.333,157.860
C02470=1031.000,-50.280,413.807,167.810,42.331,157.860
C02471=1031.006,-50.030,413.794,167.813,42.330,157.860
C02472=1031.012,-49.780,413.782,167.816,42.329,157.860
C02473=1031.018,-49.531,413.769,167.819,42.327,157.860
C02474=1031.024,-49.282,413.757,167.821,42.326,157.860
C02475=1031.030,-49.032,413.745,167.824,42.325,157.860
C02476=1031.036,-48.782,413.732,167.826,42.324,157.860
C02477=1031.042,-48.532,413.720,167.829,42.322,157.860
C02478=1031.048,-48.282,413.708,167.832,42.321,157.860
C02479=1031.055,-48.033,413.696,167.835,42.320,157.860
C02480=1031.061,-47.784,413.683,167.837,42.318,157.860
C02481=1031.067,-47.534,413.670,167.840,42.317,157.860
C02482=1031.073,-47.284,413.658,167.843,42.316,157.860
C02483=1031.079,-47.035,413.646,167.845,42.315,157.860
C02484=1031.085,-46.785,413.633,167.848,42.313,157.860
C02485=1031.091,-46.535,413.621,167.850,42.312,157.860
C02486=1031.098,-46.286,413.608,167.853,42.311,157.860
C02487=1031.104,-46.036,413.596,167.856,42.309,157.859
C02488=1031.110,-45.786,413.583,167.859,42.308,157.859
C02489=1031.116,-45.537,413.571,167.862,42.307,157.859
C02490=1031.122,-45.287,413.559,167.863,42.305,157.859
C02491=1031.128,-45.038,413.545,167.866,42.304,157.859
C02492=1031.135,-44.788,413.533,167.869,42.303,157.859
C02493=1031.141,-44.538,413.521,167.872,42.302,157.859
C02494=1031.147,-44.288,413.508,167.875,42.300,157.859
C02495=1031.154,-44.039,413.496,167.878,42.299,157.859
C02496=1031.160,-43.790,413.483,167.880,42.298,157.859
C02497=1031.166,-43.540,413.470,167.882,42.296,157.859
C02498=1031.172,-43.290,413.458,167.885,42.295,157.859
C02499=1031.178,-43.041,413.445,167.888,42.294,157.859
C02500=1031.184,-42.791,413.433,167.890,42.292,157.859
C02501=1031.190,-42.541,413.420,167.893,42.291,157.859
C02502=1031.197,-42.292,413.407,167.896,42.290,157.859
C02503=1031.203,-42.042,413.395,167.898,42.289,157.859
C02504=1031.209,-41.792,413.382,167.901,42.288,157.859
C02505=1031.216,-41.543,413.370,167.904,42.286,157.859
C02506=1031.222,-41.294,413.357,167.906,42.285,157.858
C02507=1031.228,-41.044,413.345,167.909,42.284,157.858
C02508=1031.234,-40.794,413.331,167.912,42.282,157.858
C02509=1031.241,-40.545,413.319,167.915,42.281,157.858
C02510=1031.247,-40.296,413.306,167.917,42.280,157.858
C02511=1031.253,-40.046,413.293,167.919,42.279,157.858
C02512=1031.259,-39.796,413.281,167.922,42.277,157.858
C02513=1031.266,-39.547,413.268,167.925,42.276,157.858
C02514=1031.272,-39.297,413.256,167.928,42.275,157.858
C02515=1031.278,-39.048,413.242,167.931,42.273,157.858
C02516=1031.284,-38.798,413.230,167.932,42.272,157.858
C02517=1031.290,-38.548,413.217,167.935,42.271,157.858
C02518=1031.297,-38.299,413.205,167.938,42.270,157.858
C02519=1031.303,-38.049,413.191,167.941,42.268,157.858
C02520=1031.309,-37.799,413.178,167.944,42.267,157.858
C02521=1031.315,-37.550,413.165,167.946,42.266,157.858
C02522=1031.321,-37.300,413.153,167.948,42.265,157.858
C02523=1031.328,-37.051,413.139,167.951,42.264,157.858
C02524=1031.334,-36.801,413.127,167.954,42.262,157.858
C02525=1031.341,-36.521,413.112,167.957,42.261,157.858
C02526=1031.347,-36.239,413.097,167.960,42.260,157.857
C02527=1031.354,-35.959,413.082,167.963,42.258,157.857
C02528=1031.361,-35.678,413.068,167.965,42.257,157.857
C02529=1031.367,-35.429,413.055,167.968,42.256,157.857
C02530=1031.373,-35.179,413.042,167.971,42.254,157.857
C02531=1031.380,-34.929,413.029,167.974,42.253,157.857
C02532=1031.386,-34.680,413.015,167.976,42.252,157.857
C02533=1031.392,-34.430,413.003,167.979,42.251,157.857
C02534=1031.398,-34.181,412.990,167.981,42.250,157.857
C02535=1031.404,-33.931,412.977,167.984,42.248,157.857
C02536=1031.410,-33.682,412.964,167.986,42.247,157.857
C02537=1031.417,-33.432,412.950,167.989,42.246,157.857
C02538=1031.423,-33.182,412.938,167.992,42.245,157.857
C02539=1031.429,-32.932,412.924,167.995,42.244,157.857
C02540=1031.436,-32.683,412.911,167.996,42.242,157.857
C02541=1031.442,-32.434,412.898,167.999,42.241,157.857
C02542=1031.448,-32.184,412.885,168.002,42.240,157.857
C02543=1031.455,-31.934,412.872,168.005,42.239,157.857
C02544=1031.461,-31.685,412.858,168.008,42.238,157.857
C02545=1031.467,-31.435,412.846,168.009,42.236,157.857
C02546=1031.473,-31.186,412.832,168.012,42.235,157.857
C02547=1031.479,-30.936,412.819,168.015,42.234,157.857
C02548=1031.486,-30.686,412.806,168.018,42.233,157.857
C02549=1031.492,-30.437,412.793,168.020,42.232,157.857
C02550=1031.498,-30.187,412.780,168.022,42.230,157.856
C02551=1031.504,-29.938,412.766,168.025,42.229,157.856
C02552=1031.511,-29.688,412.753,168.028,42.228,157.856
C02553=1031.517,-29.439,412.740,168.030,42.227,157.856
C02554=1031.523,-29.189,412.727,168.033,42.225,157.856
C02555=1031.529,-28.940,412.714,168.036,42.224,157.856
C02556=1031.536,-28.690,412.700,168.038,42.223,157.856
C02557=1031.542,-28.440,412.687,168.040,42.222,157.856
C02558=1031.549,-28.191,412.674,168.043,42.221,157.856
C02559=1031.555,-27.942,412.660,168.046,42.219,157.856
C02560=1031.561,-27.691,412.647,168.049,42.218,157.856
C02561=1031.568,-27.442,412.634,168.052,42.217,157.856
C02562=1031.574,-27.193,412.621,168.053,42.216,157.856
C02563=1031.580,-26.942,412.607,168.056,42.215,157.856
C02564=1031.586,-26.693,412.593,168.059,42.214,157.856
C02565=1031.592,-26.444,412.580,168.061,42.212,157.856
C02566=1031.598,-26.195,412.567,168.064,42.211,157.856
C02567=1031.605,-25.944,412.553,168.067,42.210,157.856
C02568=1031.611,-25.695,412.539,168.069,42.209,157.856
C02569=1031.617,-25.446,412.526,168.071,42.208,157.856
C02570=1031.623,-25.196,412.512,168.074,42.207,157.856
C02571=1031.629,-24.946,412.499,168.077,42.206,157.856
C02572=1031.635,-24.697,412.485,168.079,42.205,157.856
C02573=1031.642,-24.448,412.472,168.082,42.204,157.856
C02574=1031.648,-24.198,412.458,168.085,42.203,157.855
C02575=1031.654,-23.948,412.445,168.086,42.202,157.855
C02576=1031.660,-23.699,412.431,168.089,42.201,157.855
C02577=1031.666,-23.449,412.417,168.092,42.200,157.855
C02578=1031.673,-23.199,412.404,168.094,42.199,157.855
C02579=1031.679,-22.950,412.390,168.097,42.197,157.855
C02580=1031.685,-22.700,412.376,168.100,42.196,157.855
C02581=1031.691,-22.451,412.363,168.102,42.195,157.855
C02582=1031.697,-22.201,412.350,168.104,42.194,157.855
C02583=1031.704,-21.952,412.335,168.107,42.193,157.855
C02584=1031.710,-21.702,412.321,168.110,42.192,157.855
C02585=1031.717,-21.453,412.308,168.112,42.191,157.855
C02586=1031.723,-21.203,412.295,168.115,42.189,157.855
C02587=1031.728,-20.954,412.281,168.118,42.188,157.855
C02588=1031.735,-20.704,412.267,168.119,42.187,157.855
C02589=1031.742,-20.423,412.251,168.122,42.186,157.855
C02590=1031.749,-20.141,412.236,168.125,42.185,157.855
C02591=1031.756,-19.859,412.220,168.128,42.183,157.855
C02592=1031.764,-19.578,412.205,168.132,42.182,157.855
C02593=1031.769,-19.329,412.191,168.133,42.181,157.855
C02594=1031.776,-19.079,412.178,168.136,42.179,157.855
C02595=1031.782,-18.829,412.164,168.139,42.178,157.855
C02596=1031.788,-18.579,412.150,168.141,42.177,157.855
C02597=1031.795,-18.330,412.137,168.144,42.176,157.855
C02598=1031.802,-18.081,412.122,168.147,42.175,157.855
C02599=1031.807,-17.831,412.109,168.149,42.174,157.855
C02600=1031.813,-17.582,412.095,168.151,42.173,157.855
C02601=1031.820,-17.332,412.082,168.154,42.172,157.855
C02602=1031.826,-17.083,412.067,168.156,42.170,157.854
C02603=1031.833,-16.833,412.053,168.159,42.169,157.854
C02604=1031.839,-16.584,412.040,168.162,42.168,157.854
C02605=1031.845,-16.333,412.026,168.164,42.167,157.854
C02606=1031.852,-16.085,412.012,168.166,42.166,157.854
C02607=1031.859,-15.835,411.998,168.169,42.165,157.854
C02608=1031.864,-15.585,411.984,168.171,42.164,157.854
C02609=1031.871,-15.336,411.970,168.174,42.163,157.854
C02610=1031.877,-15.086,411.956,168.177,42.162,157.854
C02611=1031.883,-14.836,411.943,168.179,42.161,157.854
C02612=1031.889,-14.587,411.928,168.182,42.160,157.854
C02613=1031.895,-14.337,411.914,168.185,42.159,157.854
C02614=1031.902,-14.088,411.900,168.186,42.158,157.854
C02615=1031.908,-13.838,411.886,168.189,42.157,157.854
C02616=1031.914,-13.589,411.872,168.191,42.156,157.854
C02617=1031.920,-13.339,411.857,168.194,42.155,157.854
C02618=1031.926,-13.090,411.844,168.197,42.154,157.854
C02619=1031.933,-12.840,411.829,168.199,42.153,157.854
C02620=1031.939,-12.591,411.815,168.202,42.152,157.854
C02621=1031.946,-12.341,411.801,168.204,42.150,157.854
C02622=1031.951,-12.092,411.787,168.206,42.149,157.854
C02623=1031.958,-11.842,411.772,168.209,42.148,157.854
C02624=1031.964,-11.593,411.759,168.211,42.147,157.854
C02625=1031.970,-11.343,411.744,168.214,42.146,157.854
C02626=1031.977,-11.093,411.730,168.217,42.145,157.854
C02627=1031.983,-10.844,411.716,168.219,42.144,157.854
C02628=1031.989,-10.594,411.701,168.221,42.143,157.854
C02629=1031.995,-10.345,411.687,168.223,42.142,157.854
C02630=1032.001,-10.095,411.673,168.226,42.141,157.854
C02631=1032.008,-9.846,411.659,168.229,42.140,157.854
C02632=1032.014,-9.596,411.645,168.231,42.139,157.854
C02633=1032.020,-9.347,411.630,168.234,42.138,157.854
C02634=1032.027,-9.097,411.617,168.237,42.137,157.853
C02635=1032.033,-8.848,411.602,168.238,42.136,157.853
C02636=1032.039,-8.599,411.588,168.241,42.135,157.853
C02637=1032.046,-8.349,411.574,168.243,42.133,157.853
C02638=1032.051,-8.100,411.559,168.246,42.132,157.853
C02639=1032.058,-7.850,411.545,168.249,42.131,157.853
C02640=1032.065,-7.600,411.531,168.251,42.130,157.853
C02641=1032.070,-7.351,411.516,168.253,42.129,157.853
C02642=1032.077,-7.101,411.502,168.255,42.128,157.853
C02643=1032.084,-6.851,411.487,168.258,42.127,157.853
C02644=1032.090,-6.603,411.473,168.261,42.126,157.853
C02645=1032.096,-6.353,411.459,168.263,42.125,157.853
C02646=1032.103,-6.103,411.444,168.266,42.124,157.853
C02647=1032.109,-5.854,411.430,168.268,42.123,157.853
C02648=1032.115,-5.604,411.416,168.270,42.122,157.853
C02649=1032.121,-5.354,411.401,168.273,42.121,157.853
C02650=1032.128,-5.106,411.387,168.275,42.120,157.853
C02651=1032.134,-4.855,411.373,168.278,42.119,157.853
C02652=1032.140,-4.606,411.358,168.280,42.118,157.853
C02653=1032.148,-4.323,411.342,168.283,42.117,157.853
C02654=1032.155,-4.040,411.325,168.285,42.115,157.853
C02655=1032.162,-3.757,411.309,168.288,42.114,157.853
C02656=1032.169,-3.473,411.293,168.291,42.113,157.853
C02657=1032.176,-3.224,411.278,168.294,42.112,157.853
C02658=1032.181,-2.975,411.263,168.296,42.111,157.853
C02659=1032.188,-2.725,411.248,168.299,42.110,157.853
C02660=1032.194,-2.476,411.233,168.301,42.109,157.853
C02661=1032.200,-2.226,411.219,168.304,42.108,157.853
C02662=1032.206,-1.976,411.204,168.305,42.107,157.853
C02663=1032.212,-1.727,411.190,168.308,42.106,157.853
C02664=1032.218,-1.478,411.175,168.310,42.105,157.852
C02665=1032.225,-1.228,411.160,168.313,42.105,157.853
C02666=1032.231,-0.978,411.145,168.316,42.104,157.853
C02667=1032.237,-0.729,411.130,168.318,42.103,157.853
C02668=1032.243,-0.480,411.116,168.321,42.102,157.852
C02669=1032.249,-0.230,411.101,168.323,42.101,157.852
C02670=1032.255,0.019,411.086,168.326,42.099,157.852
C02671=1032.262,0.268,411.071,168.327,42.099,157.852
C02672=1032.268,0.519,411.057,168.330,42.097,157.852
C02673=1032.274,0.768,411.042,168.332,42.097,157.852
C02674=1032.280,1.017,411.027,168.335,42.096,157.852
C02675=1032.286,1.267,411.012,168.337,42.095,157.852
C02676=1032.293,1.517,410.997,168.340,42.094,157.852
C02677=1032.299,1.766,410.982,168.342,42.093,157.852
C02678=1032.305,2.015,410.968,168.345,42.092,157.852
C02679=1032.311,2.265,410.953,168.346,42.091,157.852
C02680=1032.318,2.515,410.938,168.349,42.090,157.852
C02681=1032.324,2.764,410.923,168.351,42.089,157.852
C02682=1032.330,3.013,410.908,168.354,42.088,157.852
C02683=1032.336,3.263,410.894,168.356,42.088,157.852
C02684=1032.343,3.513,410.879,168.359,42.087,157.852
C02685=1032.349,3.762,410.863,168.361,42.086,157.852
C02686=1032.355,4.011,410.848,168.364,42.084,157.852
C02687=1032.361,4.260,410.833,168.366,42.083,157.852
C02688=1032.368,4.510,410.818,168.368,42.082,157.852
C02689=1032.374,4.760,410.803,168.371,42.081,157.852
C02690=1032.381,5.009,410.789,168.373,42.080,157.852
C02691=1032.387,5.259,410.774,168.376,42.079,157.852
C02692=1032.393,5.508,410.759,168.378,42.078,157.852
C02693=1032.399,5.757,410.744,168.381,42.077,157.852
C02694=1032.405,6.007,410.729,168.382,42.076,157.852
C02695=1032.412,6.257,410.714,168.385,42.075,157.852
C02696=1032.419,6.506,410.699,168.387,42.075,157.852
C02697=1032.425,6.755,410.684,168.390,42.074,157.852
C02698=1032.431,7.004,410.669,168.392,42.073,157.852
C02699=1032.437,7.254,410.654,168.395,42.072,157.852
C02700=1032.443,7.504,410.639,168.397,42.071,157.852
C02701=1032.450,7.753,410.624,168.400,42.070,157.852
C02702=1032.456,8.003,410.609,168.402,42.069,157.852
C02703=1032.463,8.252,410.594,168.404,42.068,157.852
C02704=1032.469,8.502,410.579,168.406,42.067,157.852
C02705=1032.475,8.739,410.565,168.409,42.066,157.852
C02706=1032.481,8.975,410.551,168.411,42.065,157.852
C02707=1032.487,9.212,410.536,168.413,42.064,157.851
C02708=1032.493,9.448,410.522,168.416,42.063,157.851
C02709=1032.499,9.685,410.507,168.417,42.062,157.851
C02710=1032.505,9.922,410.493,168.420,42.061,157.851
C02711=1032.512,10.158,410.479,168.422,42.060,157.851
C02712=1032.517,10.395,410.465,168.424,42.059,157.851
C02713=1032.524,10.644,410.449,168.427,42.058,157.851
C02714=1032.530,10.894,410.434,168.429,42.057,157.851
C02715=1032.537,11.143,410.419,168.432,42.056,157.851
C02716=1032.543,11.393,410.404,168.434,42.055,157.851
C02717=1032.551,11.704,410.385,168.437,42.053,157.851
C02718=1032.559,12.014,410.366,168.440,42.052,157.851
C02719=1032.566,12.324,410.347,168.443,42.051,157.851
C02720=1032.575,12.635,410.328,168.446,42.050,157.851
C02721=1032.581,12.885,410.313,168.449,42.049,157.851
C02722=1032.588,13.134,410.298,168.451,42.048,157.851
C02723=1032.594,13.383,410.283,168.454,42.047,157.851
C02724=1032.601,13.633,410.268,168.455,42.046,157.851
C02725=1032.607,13.883,410.253,168.458,42.045,157.851
C02726=1032.613,14.132,410.236,168.460,42.044,157.851
C02727=1032.619,14.382,410.222,168.462,42.043,157.851
C02728=1032.626,14.631,410.206,168.465,42.042,157.851
C02729=1032.632,14.881,410.190,168.467,42.041,157.851
C02730=1032.638,15.130,410.175,168.470,42.041,157.851
C02731=1032.645,15.379,410.160,168.472,42.040,157.851
C02732=1032.650,15.629,410.144,168.474,42.039,157.851
C02733=1032.657,15.878,410.129,168.476,42.038,157.851
C02734=1032.664,16.128,410.114,168.479,42.037,157.851
C02735=1032.670,16.377,410.098,168.481,42.036,157.851
C02736=1032.676,16.627,410.082,168.484,42.035,157.851
C02737=1032.683,16.876,410.067,168.486,42.034,157.851
C02738=1032.689,17.126,410.052,168.488,42.033,157.851
C02739=1032.695,17.375,410.036,168.491,42.032,157.851
C02740=1032.702,17.624,410.020,168.492,42.031,157.851
C02741=1032.708,17.874,410.005,168.495,42.030,157.851
C02742=1032.714,18.123,409.989,168.497,42.029,157.851
C02743=1032.720,18.373,409.974,168.500,42.028,157.851
C02744=1032.727,18.622,409.958,168.502,42.027,157.850
C02745=1032.733,18.872,409.943,168.505,42.027,157.851
C02746=1032.739,19.121,409.927,168.507,42.026,157.851
C02747=1032.746,19.371,409.912,168.510,42.025,157.850
C02748=1032.752,19.620,409.896,168.512,42.024,157.850
C02749=1032.758,19.869,409.880,168.513,42.023,157.850
C02750=1032.764,20.119,409.864,168.516,42.022,157.850
C02751=1032.771,20.368,409.849,168.518,42.021,157.850
C02752=1032.777,20.617,409.833,168.521,42.020,157.850
C02753=1032.783,20.867,409.818,168.523,42.020,157.850
C02754=1032.789,21.116,409.801,168.526,42.018,157.850
C02755=1032.796,21.366,409.785,168.528,42.018,157.850
C02756=1032.803,21.616,409.770,168.530,42.017,157.850
C02757=1032.809,21.865,409.754,168.533,42.016,157.850
C02758=1032.815,22.114,409.738,168.534,42.015,157.850
C02759=1032.821,22.364,409.723,168.537,42.014,157.850
C02760=1032.828,22.613,409.707,168.539,42.013,157.850
C02761=1032.834,22.862,409.691,168.542,42.012,157.850
C02762=1032.840,23.112,409.676,168.544,42.011,157.850
C02763=1032.846,23.361,409.660,168.546,42.011,157.850
C02764=1032.853,23.611,409.644,168.549,42.010,157.850
C02765=1032.859,23.860,409.628,168.551,42.009,157.850
C02766=1032.865,24.110,409.613,168.553,42.008,157.850
C02767=1032.871,24.360,409.596,168.555,42.007,157.850
C02768=1032.878,24.609,409.581,168.558,42.006,157.850
C02769=1032.884,24.858,409.564,168.560,42.005,157.850
C02770=1032.891,25.108,409.549,168.562,42.005,157.850
C02771=1032.896,25.357,409.533,168.565,42.003,157.850
C02772=1032.903,25.606,409.517,168.567,42.002,157.850
C02773=1032.909,25.855,409.501,168.570,42.001,157.850
C02774=1032.916,26.105,409.485,168.571,42.000,157.850
C02775=1032.922,26.354,409.469,168.574,41.999,157.850
C02776=1032.929,26.604,409.454,168.576,41.998,157.850
C02777=1032.935,26.853,409.438,168.578,41.998,157.850
C02778=1032.941,27.102,409.422,168.581,41.997,157.850
C02779=1032.947,27.352,409.406,168.583,41.996,157.850
C02780=1032.953,27.601,409.390,168.586,41.995,157.850
C02781=1032.961,27.888,409.372,168.588,41.994,157.850
C02782=1032.968,28.174,409.354,168.591,41.993,157.850
C02783=1032.975,28.461,409.334,168.593,41.992,157.850
C02784=1032.983,28.747,409.316,168.596,41.991,157.850
C02785=1032.989,28.996,409.300,168.598,41.991,157.850
C02786=1032.995,29.245,409.284,168.600,41.990,157.850
C02787=1033.002,29.495,409.267,168.603,41.989,157.850
C02788=1033.008,29.745,409.251,168.605,41.988,157.850
C02789=1033.014,29.994,409.235,168.608,41.987,157.850
C02790=1033.020,30.243,409.219,168.610,41.986,157.850
C02791=1033.026,30.492,409.203,168.612,41.985,157.850
C02792=1033.033,30.741,409.187,168.614,41.984,157.850
C02793=1033.040,30.991,409.170,168.616,41.983,157.850
C02794=1033.045,31.241,409.154,168.618,41.983,157.850
C02795=1033.051,31.490,409.138,168.621,41.982,157.850
C02796=1033.058,31.739,409.122,168.623,41.981,157.850
C02797=1033.064,31.988,409.106,168.626,41.980,157.850
C02798=1033.071,32.239,409.089,168.628,41.980,157.850
C02799=1033.077,32.488,409.073,168.630,41.979,157.850
C02800=1033.083,32.737,409.057,168.633,41.978,157.850
C02801=1033.089,32.986,409.041,168.635,41.977,157.849
C02802=1033.096,33.236,409.025,168.637,41.976,157.849
C02803=1033.102,33.486,409.008,168.639,41.975,157.850
C02804=1033.108,33.735,408.993,168.641,41.974,157.849
C02805=1033.114,33.984,408.976,168.644,41.973,157.849
C02806=1033.121,34.234,408.960,168.646,41.972,157.849
C02807=1033.127,34.483,408.944,168.648,41.971,157.849
C02808=1033.134,34.732,408.927,168.651,41.971,157.849
C02809=1033.140,34.981,408.911,168.653,41.970,157.849
C02810=1033.146,35.231,408.894,168.656,41.969,157.849
C02811=1033.152,35.481,408.878,168.657,41.968,157.849
C02812=1033.159,35.730,408.862,168.659,41.967,157.849
C02813=1033.166,35.980,408.846,168.662,41.966,157.849
C02814=1033.171,36.229,408.830,168.664,41.966,157.849
C02815=1033.178,36.478,408.813,168.667,41.965,157.849
C02816=1033.184,36.727,408.797,168.669,41.964,157.849
C02817=1033.191,36.977,408.780,168.671,41.963,157.849
C02818=1033.197,37.226,408.764,168.674,41.962,157.849
C02819=1033.203,37.476,408.748,168.676,41.961,157.849
C02820=1033.210,37.725,408.730,168.677,41.960,157.849
C02821=1033.216,37.974,408.714,168.680,41.959,157.849
C02822=1033.222,38.224,408.698,168.682,41.958,157.849
C02823=1033.229,38.473,408.681,168.684,41.958,157.849
C02824=1033.234,38.722,408.664,168.687,41.957,157.849
C02825=1033.240,38.972,408.648,168.689,41.956,157.849
C02826=1033.247,39.222,408.631,168.692,41.956,157.849
C02827=1033.253,39.471,408.614,168.694,41.955,157.849
C02828=1033.259,39.720,408.598,168.696,41.954,157.849
C02829=1033.265,39.969,408.582,168.699,41.953,157.849
C02830=1033.272,40.219,408.565,168.701,41.952,157.849
C02831=1033.278,40.468,408.548,168.702,41.951,157.849
C02832=1033.284,40.717,408.532,168.705,41.950,157.849
C02833=1033.291,40.967,408.515,168.707,41.949,157.849
C02834=1033.297,41.216,408.498,168.709,41.949,157.849
C02835=1033.304,41.466,408.481,168.712,41.948,157.849
C02836=1033.310,41.715,408.465,168.714,41.947,157.849
C02837=1033.315,41.964,408.449,168.716,41.946,157.849
C02838=1033.322,42.214,408.431,168.719,41.946,157.849
C02839=1033.328,42.463,408.415,168.721,41.945,157.849
C02840=1033.334,42.712,408.399,168.722,41.944,157.849
C02841=1033.341,42.962,408.381,168.725,41.943,157.849
C02842=1033.347,43.211,408.365,168.727,41.943,157.849
C02843=1033.354,43.461,408.348,168.729,41.942,157.849
C02844=1033.360,43.710,408.332,168.732,41.941,157.849
C02845=1033.367,43.996,408.312,168.734,41.940,157.849
C02846=1033.373,44.282,408.292,168.737,41.939,157.849
C02847=1033.381,44.568,408.273,168.740,41.938,157.849
C02848=1033.388,44.855,408.254,168.742,41.938,157.849
C02849=1033.395,45.104,408.236,168.745,41.937,157.849
C02850=1033.400,45.354,408.220,168.747,41.936,157.849
C02851=1033.406,45.602,408.203,168.749,41.936,157.849
C02852=1033.413,45.853,408.186,168.750,41.935,157.849
C02853=1033.418,46.102,408.168,168.754,41.934,157.849
C02854=1033.425,46.352,408.152,168.755,41.933,157.849
C02855=1033.431,46.600,408.135,168.757,41.932,157.849
C02856=1033.437,46.849,408.118,168.760,41.932,157.849
C02857=1033.443,47.099,408.101,168.762,41.931,157.849
C02858=1033.449,47.348,408.084,168.764,41.930,157.849
C02859=1033.456,47.598,408.067,168.767,41.930,157.849
C02860=1033.462,47.847,408.050,168.769,41.929,157.849
C02861=1033.468,48.097,408.032,168.771,41.928,157.849
C02862=1033.474,48.346,408.016,168.774,41.927,157.849
C02863=1033.480,48.595,407.999,168.776,41.926,157.849
C02864=1033.487,48.845,407.981,168.777,41.925,157.849
C02865=1033.493,49.094,407.965,168.779,41.925,157.849
C02866=1033.499,49.343,407.947,168.782,41.924,157.849
C02867=1033.506,49.592,407.930,168.784,41.923,157.849
C02868=1033.511,49.842,407.913,168.786,41.923,157.849
C02869=1033.518,50.091,407.896,168.789,41.922,157.849
C02870=1033.525,50.341,407.879,168.791,41.921,157.849
C02871=1033.530,50.590,407.862,168.793,41.921,157.849
C02872=1033.536,50.839,407.845,168.796,41.920,157.849
C02873=1033.543,51.088,407.828,168.798,41.919,157.849
C02874=1033.549,51.338,407.811,168.800,41.918,157.849
C02875=1033.555,51.587,407.794,168.803,41.917,157.849
C02876=1033.561,51.836,407.777,168.804,41.916,157.849
C02877=1033.568,52.086,407.759,168.806,41.916,157.849
C02878=1033.573,52.335,407.742,168.809,41.915,157.849
C02879=1033.580,52.585,407.725,168.811,41.914,157.849
C02880=1033.586,52.833,407.708,168.813,41.914,157.849
C02881=1033.593,53.083,407.691,168.815,41.913,157.849
C02882=1033.599,53.333,407.673,168.818,41.912,157.849
C02883=1033.605,53.582,407.657,168.820,41.911,157.849
C02884=1033.612,53.831,407.639,168.822,41.910,157.849
C02885=1033.618,54.080,407.622,168.825,41.909,157.849
C02886=1033.625,54.330,407.604,168.826,41.908,157.849
C02887=1033.631,54.579,407.587,168.829,41.908,157.849
C02888=1033.637,54.829,407.570,168.831,41.907,157.849
C02889=1033.643,55.078,407.553,168.833,41.906,157.849
C02890=1033.650,55.327,407.536,168.835,41.905,157.849
C02891=1033.655,55.576,407.518,168.838,41.905,157.849
C02892=1033.662,55.826,407.501,168.840,41.904,157.849
C02893=1033.669,56.075,407.484,168.842,41.903,157.849
C02894=1033.674,56.325,407.467,168.845,41.902,157.849
C02895=1033.681,56.574,407.449,168.847,41.902,157.849
C02896=1033.687,56.823,407.432,168.849,41.901,157.849
C02897=1033.694,57.072,407.415,168.851,41.900,157.849
C02898=1033.700,57.322,407.397,168.853,41.899,157.849
C02899=1033.707,57.571,407.380,168.855,41.898,157.849
C02900=1033.713,57.820,407.363,168.858,41.897,157.849
C02901=1033.719,58.069,407.345,168.860,41.896,157.849
C02902=1033.726,58.319,407.328,168.862,41.895,157.848
C02903=1033.732,58.569,407.311,168.865,41.895,157.849
C02904=1033.738,58.818,407.294,168.867,41.894,157.848
C02905=1033.745,59.067,407.276,168.869,41.893,157.848
C02906=1033.751,59.316,407.259,168.871,41.892,157.848
C02907=1033.757,59.566,407.241,168.874,41.892,157.848
C02908=1033.764,59.815,407.224,168.875,41.891,157.848
C02909=1033.771,60.101,407.204,168.878,41.890,157.848
C02910=1033.778,60.387,407.184,168.881,41.889,157.848
C02911=1033.786,60.673,407.165,168.883,41.888,157.848
C02912=1033.793,60.959,407.144,168.886,41.887,157.848
C02913=1033.800,61.208,407.127,168.888,41.886,157.848
C02914=1033.806,61.457,407.109,168.891,41.885,157.848
C02915=1033.813,61.706,407.092,168.893,41.884,157.848
C02916=1033.820,61.956,407.074,168.894,41.883,157.848
C02917=1033.825,62.205,407.057,168.897,41.882,157.848
C02918=1033.832,62.454,407.039,168.899,41.881,157.848
C02919=1033.838,62.704,407.021,168.901,41.881,157.848
C02920=1033.844,62.953,407.004,168.904,41.880,157.848
C02921=1033.851,63.202,406.987,168.906,41.879,157.848
C02922=1033.857,63.452,406.969,168.909,41.878,157.848
C02923=1033.864,63.701,406.952,168.911,41.877,157.848
C02924=1033.870,63.950,406.934,168.913,41.877,157.848
C02925=1033.877,64.200,406.917,168.914,41.876,157.848
C02926=1033.883,64.450,406.899,168.917,41.876,157.848
C02927=1033.889,64.698,406.881,168.919,41.875,157.848
C02928=1033.895,64.947,406.863,168.921,41.874,157.848
C02929=1033.901,65.197,406.845,168.924,41.873,157.848
C02930=1033.908,65.446,406.828,168.926,41.872,157.848
C02931=1033.914,65.696,406.811,168.928,41.871,157.848
C02932=1033.920,65.945,406.793,168.931,41.871,157.848
C02933=1033.927,66.194,406.775,168.933,41.870,157.848
C02934=1033.933,66.443,406.757,168.935,41.869,157.848
C02935=1033.939,66.693,406.739,168.937,41.869,157.848
C02936=1033.946,66.942,406.722,168.940,41.868,157.848
C02937=1033.951,67.191,406.703,168.941,41.867,157.848
C02938=1033.958,67.441,406.686,168.943,41.867,157.848
C02939=1033.964,67.690,406.668,168.946,41.865,157.848
C02940=1033.970,67.939,406.651,168.948,41.865,157.848
C02941=1033.976,68.188,406.632,168.950,41.864,157.848
C02942=1033.983,68.438,406.615,168.952,41.863,157.848
C02943=1033.989,68.687,406.597,168.955,41.862,157.848
C02944=1033.995,68.936,406.578,168.957,41.862,157.848
C02945=1034.001,69.186,406.560,168.959,41.861,157.848
C02946=1034.008,69.435,406.543,168.962,41.860,157.848
C02947=1034.015,69.684,406.524,168.964,41.860,157.848
C02948=1034.020,69.933,406.507,168.965,41.859,157.848
C02949=1034.026,70.183,406.489,168.968,41.859,157.848
C02950=1034.033,70.432,406.470,168.970,41.857,157.848
C02951=1034.040,70.681,406.453,168.972,41.857,157.848
C02952=1034.045,70.930,406.435,168.974,41.856,157.848
C02953=1034.051,71.180,406.417,168.977,41.855,157.848
C02954=1034.058,71.429,406.399,168.979,41.855,157.848
C02955=1034.064,71.678,406.380,168.981,41.854,157.848
C02956=1034.070,71.928,406.362,168.983,41.853,157.848
C02957=1034.077,72.176,406.345,168.986,41.853,157.848
C02958=1034.083,72.426,406.327,168.988,41.852,157.848
C02959=1034.089,72.675,406.308,168.990,41.851,157.848
C02960=1034.095,72.925,406.290,168.993,41.850,157.848
C02961=1034.101,73.174,406.273,168.994,41.849,157.848
C02962=1034.107,73.423,406.254,168.997,41.849,157.848
C02963=1034.113,73.673,406.236,168.998,41.848,157.848
C02964=1034.120,73.922,406.217,169.001,41.847,157.848
C02965=1034.127,74.171,406.200,169.003,41.847,157.848
C02966=1034.133,74.420,406.182,169.005,41.846,157.848
C02967=1034.139,74.670,406.164,169.008,41.845,157.848
C02968=1034.145,74.919,406.145,169.010,41.845,157.848
C02969=1034.151,75.168,406.127,169.012,41.844,157.848
C02970=1034.158,75.417,406.108,169.015,41.843,157.848
C02971=1034.164,75.667,406.090,169.017,41.842,157.848
C02972=1034.170,75.915,406.073,169.019,41.841,157.848
C02973=1034.177,76.202,406.051,169.022,41.841,157.848
C02974=1034.185,76.487,406.031,169.023,41.840,157.848
C02975=1034.193,76.773,406.010,169.026,41.839,157.848
C02976=1034.199,77.059,405.989,169.029,41.838,157.848
C02977=1034.205,77.308,405.970,169.031,41.838,157.848
C02978=1034.212,77.557,405.952,169.033,41.837,157.848
C02979=1034.218,77.807,405.934,169.035,41.836,157.848
C02980=1034.224,78.056,405.915,169.038,41.835,157.848
C02981=1034.230,78.305,405.897,169.040,41.835,157.848
C02982=1034.236,78.554,405.879,169.042,41.834,157.848
C02983=1034.243,78.804,405.860,169.045,41.834,157.848
C02984=1034.249,79.053,405.842,169.047,41.833,157.848
C02985=1034.254,79.303,405.823,169.049,41.832,157.848
C02986=1034.261,79.552,405.804,169.051,41.832,157.848
C02987=1034.267,79.801,405.786,169.053,41.830,157.848
C02988=1034.273,80.050,405.768,169.056,41.830,157.848
C02989=1034.279,80.299,405.750,169.057,41.829,157.848
C02990=1034.286,80.548,405.731,169.059,41.829,157.848
C02991=1034.292,80.797,405.712,169.062,41.828,157.848
C02992=1034.297,81.048,405.694,169.064,41.828,157.848
C02993=1034.304,81.297,405.675,169.066,41.827,157.848
C02994=1034.310,81.546,405.656,169.069,41.826,157.848
C02995=1034.317,81.795,405.638,169.071,41.825,157.848
C02996=1034.323,82.043,405.620,169.073,41.825,157.848
C02997=1034.329,82.293,405.602,169.075,41.824,157.848
C02998=1034.335,82.542,405.583,169.078,41.824,157.848
C02999=1034.341,82.792,405.564,169.080,41.823,157.848
C03000=1034.347,83.041,405.545,169.082,41.822,157.848
C03001=1034.354,83.290,405.526,169.084,41.822,157.848
C03002=1034.360,83.540,405.508,169.087,41.821,157.848
C03003=1034.366,83.789,405.490,169.089,41.820,157.848
C03004=1034.373,84.038,405.471,169.090,41.819,157.848
C03005=1034.378,84.287,405.452,169.093,41.819,157.848
C03006=1034.385,84.536,405.433,169.095,41.818,157.848
C03007=1034.391,84.785,405.415,169.097,41.817,157.848
C03008=1034.398,85.035,405.396,169.099,41.817,157.848
C03009=1034.404,85.284,405.378,169.102,41.816,157.848
C03010=1034.410,85.533,405.359,169.104,41.815,157.848
C03011=1034.416,85.783,405.340,169.106,41.815,157.848
C03012=1034.422,86.032,405.322,169.109,41.814,157.848
C03013=1034.429,86.281,405.303,169.111,41.813,157.848
C03014=1034.435,86.530,405.284,169.113,41.812,157.848
C03015=1034.441,86.779,405.266,169.116,41.812,157.848
C03016=1034.448,87.029,405.247,169.118,41.811,157.848
C03017=1034.454,87.278,405.228,169.120,41.811,157.848
C03018=1034.460,87.527,405.209,169.121,41.810,157.848
C03019=1034.466,87.776,405.190,169.124,41.809,157.848
C03020=1034.473,88.025,405.172,169.126,41.808,157.848
C03021=1034.479,88.274,405.153,169.128,41.807,157.848
C03022=1034.486,88.524,405.134,169.131,41.807,157.848
C03023=1034.491,88.773,405.115,169.133,41.806,157.848
C03024=1034.498,89.022,405.097,169.135,41.805,157.848
C03025=1034.504,89.271,405.078,169.138,41.805,157.848
C03026=1034.511,89.520,405.059,169.140,41.804,157.848
C03027=1034.517,89.769,405.041,169.142,41.803,157.848
C03028=1034.523,90.019,405.021,169.145,41.803,157.848
C03029=1034.529,90.268,405.003,169.147,41.802,157.848
C03030=1034.535,90.517,404.983,169.149,41.801,157.848
C03031=1034.541,90.767,404.965,169.151,41.801,157.848
C03032=1034.547,91.016,404.946,169.153,41.800,157.848
C03033=1034.553,91.265,404.927,169.155,41.800,157.848
C03034=1034.559,91.515,404.908,169.157,41.799,157.848
C03035=1034.566,91.764,404.889,169.159,41.798,157.848
C03036=1034.572,92.012,404.870,169.162,41.797,157.848
C03037=1034.579,92.299,404.848,169.164,41.797,157.848
C03038=1034.586,92.584,404.826,169.167,41.796,157.848
C03039=1034.593,92.870,404.804,169.170,41.796,157.848
C03040=1034.601,93.156,404.782,169.172,41.795,157.848
C03041=1034.607,93.405,404.763,169.174,41.794,157.848
C03042=1034.613,93.654,404.744,169.177,41.793,157.848
C03043=1034.619,93.904,404.725,169.179,41.792,157.848
C03044=1034.625,94.153,404.706,169.181,41.792,157.848
C03045=1034.631,94.401,404.686,169.184,41.792,157.848
C03046=1034.638,94.651,404.668,169.186,41.791,157.848
C03047=1034.643,94.900,404.648,169.188,41.791,157.848
C03048=1034.650,95.149,404.630,169.190,41.790,157.848
C03049=1034.656,95.398,404.610,169.192,41.789,157.848
C03050=1034.662,95.647,404.591,169.194,41.788,157.848
C03051=1034.668,95.897,404.572,169.196,41.787,157.848
C03052=1034.675,96.146,404.553,169.199,41.787,157.849
C03053=1034.681,96.395,404.533,169.201,41.786,157.848
C03054=1034.687,96.644,404.514,169.203,41.786,157.849
C03055=1034.693,96.894,404.495,169.206,41.785,157.848
C03056=1034.699,97.143,404.476,169.208,41.784,157.849
C03057=1034.705,97.392,404.456,169.210,41.784,157.848
C03058=1034.712,97.641,404.438,169.212,41.783,157.849
C03059=1034.717,97.890,404.419,169.215,41.782,157.849
C03060=1034.725,98.139,404.399,169.217,41.782,157.849
C03061=1034.730,98.389,404.380,169.219,41.781,157.849
C03062=1034.737,98.638,404.361,169.222,41.781,157.849
C03063=1034.743,98.887,404.341,169.224,41.780,157.849
C03064=1034.749,99.136,404.322,169.226,41.779,157.849
C03065=1034.755,99.385,404.303,169.228,41.778,157.849
C03066=1034.762,99.635,404.283,169.230,41.778,157.849
C03067=1034.768,99.884,404.264,169.232,41.777,157.849
C03068=1034.775,100.132,404.245,169.235,41.776,157.849
C03069=1034.780,100.382,404.226,169.237,41.776,157.849
C03070=1034.786,100.631,404.206,169.239,41.775,157.849
C03071=1034.793,100.880,404.187,169.241,41.775,157.849
C03072=1034.798,101.129,404.168,169.244,41.774,157.849
C03073=1034.805,101.379,404.147,169.246,41.774,157.849
C03074=1034.811,101.628,404.128,169.248,41.773,157.849
C03075=1034.817,101.877,404.108,169.251,41.773,157.849
C03076=1034.823,102.126,404.089,169.253,41.772,157.849
C03077=1034.829,102.375,404.070,169.255,41.771,157.849
C03078=1034.835,102.624,404.050,169.257,41.770,157.849
C03079=1034.841,102.874,404.030,169.260,41.770,157.849
C03080=1034.848,103.122,404.011,169.262,41.770,157.849
C03081=1034.854,103.372,403.991,169.264,41.769,157.849
C03082=1034.860,103.621,403.971,169.267,41.768,157.849
C03083=1034.866,103.870,403.952,169.269,41.767,157.849
C03084=1034.873,104.119,403.932,169.271,41.767,157.849
C03085=1034.879,104.369,403.913,169.273,41.767,157.849
C03086=1034.885,104.618,403.893,169.275,41.766,157.849
C03087=1034.891,104.866,403.873,169.278,41.766,157.849
C03088=1034.896,105.116,403.854,169.279,41.765,157.849
C03089=1034.904,105.365,403.834,169.282,41.764,157.849
C03090=1034.909,105.614,403.815,169.284,41.763,157.849
C03091=1034.915,105.863,403.795,169.286,41.763,157.849
C03092=1034.921,106.112,403.775,169.289,41.763,157.849
C03093=1034.928,106.362,403.756,169.291,41.762,157.849
C03094=1034.934,106.611,403.736,169.293,41.761,157.849
C03095=1034.940,106.859,403.716,169.296,41.760,157.849
C03096=1034.946,107.109,403.697,169.298,41.760,157.849
C03097=1034.953,107.358,403.677,169.300,41.759,157.849
C03098=1034.959,107.608,403.658,169.303,41.759,157.849
C03099=1034.965,107.856,403.638,169.305,41.758,157.849
C03100=1034.972,108.106,403.618,169.307,41.758,157.849
C03101=1034.978,108.391,403.596,169.310,41.756,157.849
C03102=1034.985,108.677,403.573,169.313,41.756,157.849
C03103=1034.993,108.963,403.550,169.315,41.755,157.849
C03104=1034.999,109.249,403.527,169.318,41.755,157.849
C03105=1035.006,109.498,403.507,169.319,41.754,157.849
C03106=1035.013,109.747,403.488,169.323,41.753,157.849
C03107=1035.018,109.996,403.469,169.324,41.752,157.849
C03108=1035.025,110.246,403.448,169.326,41.752,157.849
C03109=1035.031,110.494,403.428,169.329,41.752,157.850
C03110=1035.037,110.743,403.408,169.331,41.751,157.850
C03111=1035.043,110.993,403.388,169.333,41.751,157.850
C03112=1035.049,111.242,403.369,169.336,41.750,157.850
C03113=1035.055,111.491,403.349,169.338,41.749,157.850
C03114=1035.062,111.740,403.328,169.340,41.749,157.850
C03115=1035.068,111.989,403.309,169.343,41.748,157.850
C03116=1035.074,112.238,403.289,169.345,41.748,157.850
C03117=1035.080,112.488,403.268,169.347,41.747,157.850
C03118=1035.086,112.737,403.249,169.350,41.746,157.850
C03119=1035.092,112.986,403.229,169.352,41.746,157.850
C03120=1035.099,113.235,403.209,169.354,41.745,157.850
C03121=1035.105,113.484,403.189,169.356,41.745,157.850
C03122=1035.111,113.733,403.169,169.359,41.744,157.850
C03123=1035.117,113.983,403.148,169.361,41.744,157.850
C03124=1035.123,114.231,403.128,169.363,41.743,157.850
C03125=1035.128,114.480,403.108,169.366,41.743,157.850
C03126=1035.135,114.730,403.088,169.368,41.743,157.850
C03127=1035.141,114.979,403.068,169.370,41.742,157.850
C03128=1035.147,115.228,403.048,169.373,41.741,157.850
C03129=1035.152,115.477,403.027,169.375,41.741,157.850
C03130=1035.159,115.726,403.007,169.377,41.741,157.850
C03131=1035.165,115.975,402.987,169.379,41.740,157.850
C03132=1035.171,116.225,402.967,169.382,41.739,157.850
C03133=1035.177,116.474,402.946,169.384,41.739,157.850
C03134=1035.183,116.722,402.926,169.386,41.739,157.850
C03135=1035.189,116.972,402.906,169.389,41.738,157.850
C03136=1035.195,117.221,402.886,169.391,41.737,157.851
C03137=1035.201,117.470,402.865,169.393,41.737,157.851
C03138=1035.207,117.719,402.844,169.396,41.737,157.851
C03139=1035.213,117.968,402.824,169.398,41.736,157.851
C03140=1035.219,118.216,402.804,169.400,41.736,157.851
C03141=1035.225,118.466,402.783,169.403,41.735,157.851
C03142=1035.231,118.715,402.763,169.404,41.734,157.851
C03143=1035.238,118.965,402.743,169.407,41.734,157.851
C03144=1035.244,119.213,402.723,169.410,41.734,157.851
C03145=1035.249,119.463,402.703,169.412,41.733,157.851
C03146=1035.256,119.712,402.682,169.413,41.732,157.851
C03147=1035.262,119.960,402.662,169.416,41.732,157.851
C03148=1035.269,120.210,402.641,169.418,41.732,157.851
C03149=1035.274,120.459,402.621,169.420,41.731,157.851
C03150=1035.280,120.708,402.600,169.423,41.730,157.851
C03151=1035.286,120.957,402.580,169.425,41.730,157.851
C03152=1035.292,121.206,402.559,169.427,41.729,157.851
C03153=1035.299,121.455,402.539,169.430,41.729,157.851
C03154=1035.305,121.704,402.519,169.432,41.728,157.851
C03155=1035.311,121.954,402.498,169.434,41.728,157.851
C03156=1035.316,122.203,402.478,169.437,41.727,157.851
C03157=1035.323,122.452,402.457,169.439,41.727,157.851
C03158=1035.329,122.700,402.437,169.442,41.726,157.851
C03159=1035.336,122.950,402.417,169.444,41.726,157.851
C03160=1035.341,123.199,402.396,169.446,41.725,157.851
C03161=1035.348,123.448,402.375,169.449,41.725,157.852
C03162=1035.354,123.697,402.355,169.451,41.724,157.851
C03163=1035.360,123.947,402.334,169.453,41.724,157.852
C03164=1035.366,124.195,402.314,169.456,41.723,157.852
C03165=1035.373,124.481,402.290,169.459,41.722,157.852
C03166=1035.380,124.766,402.267,169.461,41.722,157.852
C03167=1035.387,125.052,402.243,169.464,41.722,157.852
C03168=1035.395,125.338,402.219,169.467,41.720,157.852
C03169=1035.401,125.586,402.199,169.469,41.720,157.852
C03170=1035.407,125.835,402.178,169.472,41.720,157.852
C03171=1035.413,126.084,402.158,169.474,41.719,157.852
C03172=1035.419,126.334,402.137,169.476,41.719,157.852
C03173=1035.426,126.582,402.117,169.479,41.718,157.852
C03174=1035.432,126.832,402.096,169.481,41.717,157.852
C03175=1035.437,127.081,402.076,169.483,41.717,157.852
C03176=1035.444,127.330,402.055,169.486,41.717,157.852
C03177=1035.451,127.579,402.034,169.488,41.716,157.852
C03178=1035.456,127.828,402.014,169.491,41.715,157.852
C03179=1035.463,128.077,401.993,169.493,41.715,157.852
C03180=1035.469,128.326,401.973,169.496,41.714,157.852
C03181=1035.476,128.575,401.952,169.498,41.714,157.852
C03182=1035.481,128.824,401.931,169.500,41.713,157.852
C03183=1035.488,129.073,401.910,169.502,41.712,157.852
C03184=1035.495,129.323,401.890,169.504,41.712,157.852
C03185=1035.500,129.572,401.869,169.508,41.712,157.852
C03186=1035.507,129.821,401.848,169.509,41.711,157.852
C03187=1035.514,130.070,401.828,169.511,41.710,157.852
C03188=1035.519,130.319,401.807,169.514,41.710,157.853
C03189=1035.526,130.568,401.786,169.516,41.709,157.853
C03190=1035.532,130.816,401.766,169.519,41.709,157.853
C03191=1035.538,131.066,401.745,169.521,41.708,157.853
C03192=1035.544,131.315,401.723,169.524,41.708,157.853
C03193=1035.550,131.563,401.702,169.526,41.708,157.853
C03194=1035.556,131.813,401.682,169.528,41.707,157.853
C03195=1035.562,132.061,401.661,169.531,41.706,157.853
C03196=1035.568,132.311,401.640,169.533,41.706,157.853
C03197=1035.574,132.561,401.618,169.536,41.706,157.853
C03198=1035.581,132.809,401.598,169.538,41.705,157.853
C03199=1035.587,133.059,401.577,169.540,41.705,157.853
C03200=1035.592,133.307,401.555,169.543,41.704,157.853
C03201=1035.599,133.556,401.534,169.545,41.704,157.853
C03202=1035.605,133.806,401.513,169.548,41.703,157.853
C03203=1035.611,134.054,401.492,169.550,41.703,157.853
C03204=1035.617,134.303,401.471,169.552,41.703,157.853
C03205=1035.623,134.553,401.450,169.555,41.702,157.853
C03206=1035.630,134.801,401.430,169.557,41.702,157.853
C03207=1035.636,135.050,401.408,169.560,41.701,157.854
C03208=1035.642,135.300,401.387,169.562,41.701,157.854
C03209=1035.648,135.548,401.366,169.564,41.701,157.854
C03210=1035.654,135.798,401.345,169.567,41.700,157.854
C03211=1035.660,136.047,401.323,169.569,41.699,157.854
C03212=1035.666,136.296,401.303,169.572,41.699,157.854
C03213=1035.672,136.545,401.281,169.574,41.699,157.854
C03214=1035.679,136.794,401.260,169.577,41.698,157.854
C03215=1035.685,137.042,401.239,169.579,41.698,157.854
C03216=1035.691,137.292,401.218,169.581,41.697,157.854
C03217=1035.697,137.541,401.197,169.584,41.697,157.854
C03218=1035.702,137.790,401.175,169.586,41.696,157.854
C03219=1035.709,138.039,401.154,169.589,41.696,157.854
C03220=1035.716,138.288,401.133,169.591,41.696,157.854
C03221=1035.722,138.537,401.111,169.594,41.695,157.854
C03222=1035.728,138.786,401.091,169.596,41.695,157.855
C03223=1035.734,139.035,401.069,169.598,41.694,157.854
C03224=1035.740,139.284,401.048,169.601,41.694,157.855
C03225=1035.746,139.533,401.027,169.603,41.693,157.855
C03226=1035.752,139.782,401.005,169.606,41.693,157.855
C03227=1035.758,140.031,400.983,169.608,41.693,157.855
C03228=1035.764,140.280,400.962,169.611,41.692,157.855
C03229=1035.771,140.565,400.937,169.613,41.692,157.855
C03230=1035.778,140.851,400.913,169.616,41.692,157.855
C03231=1035.785,141.136,400.889,169.620,41.691,157.855
C03232=1035.792,141.422,400.864,169.623,41.691,157.855
C03233=1035.797,141.671,400.843,169.625,41.690,157.855
C03234=1035.804,141.920,400.821,169.628,41.690,157.855
C03235=1035.810,142.169,400.799,169.629,41.689,157.855
C03236=1035.817,142.418,400.778,169.633,41.689,157.855
C03237=1035.822,142.666,400.757,169.635,41.688,157.856
C03238=1035.829,142.915,400.735,169.638,41.688,157.856
C03239=1035.835,143.164,400.713,169.640,41.688,157.856
C03240=1035.841,143.413,400.692,169.642,41.688,157.856
C03241=1035.847,143.663,400.670,169.645,41.687,157.856
C03242=1035.853,143.911,400.649,169.647,41.687,157.856
C03243=1035.859,144.160,400.627,169.650,41.686,157.856
C03244=1035.865,144.410,400.605,169.652,41.686,157.856
C03245=1035.871,144.659,400.584,169.655,41.686,157.856
C03246=1035.877,144.908,400.562,169.657,41.685,157.856
C03247=1035.884,145.156,400.541,169.660,41.685,157.856
C03248=1035.890,145.405,400.520,169.662,41.684,157.856
C03249=1035.896,145.655,400.498,169.665,41.684,157.856
C03250=1035.902,145.904,400.477,169.667,41.683,157.856
C03251=1035.909,146.152,400.454,169.670,41.683,157.857
C03252=1035.915,146.402,400.433,169.672,41.683,157.857
C03253=1035.920,146.650,400.411,169.675,41.682,157.857
C03254=1035.926,146.899,400.390,169.677,41.682,157.857
C03255=1035.933,147.148,400.368,169.680,41.682,157.857
C03256=1035.939,147.398,400.346,169.682,41.681,157.857
C03257=1035.945,147.646,400.324,169.685,41.681,157.857
C03258=1035.951,147.895,400.302,169.687,41.681,157.857
C03259=1035.957,148.144,400.281,169.690,41.680,157.857
C03260=1035.962,148.393,400.259,169.692,41.680,157.857
C03261=1035.969,148.642,400.237,169.695,41.680,157.857
C03262=1035.975,148.891,400.215,169.697,41.679,157.857
C03263=1035.981,149.140,400.193,169.699,41.679,157.858
C03264=1035.988,149.389,400.171,169.702,41.679,157.858
C03265=1035.994,149.638,400.149,169.704,41.678,157.858
C03266=1035.999,149.887,400.128,169.707,41.678,157.858
C03267=1036.006,150.136,400.106,169.709,41.678,157.858
C03268=1036.011,150.385,400.083,169.712,41.677,157.858
C03269=1036.017,150.634,400.062,169.714,41.677,157.858
C03270=1036.024,150.883,400.040,169.717,41.677,157.858
C03271=1036.030,151.132,400.018,169.719,41.676,157.858
C03272=1036.036,151.381,399.996,169.722,41.676,157.858
C03273=1036.042,151.630,399.973,169.724,41.676,157.858
C03274=1036.048,151.879,399.952,169.728,41.676,157.859
C03275=1036.054,152.128,399.930,169.730,41.676,157.859
C03276=1036.060,152.376,399.908,169.733,41.675,157.859
C03277=1036.066,152.625,399.886,169.736,41.675,157.859
C03278=1036.072,152.874,399.863,169.738,41.675,157.859
C03279=1036.078,153.124,399.842,169.741,41.674,157.859
C03280=1036.085,153.372,399.819,169.743,41.674,157.859
C03281=1036.091,153.621,399.798,169.746,41.673,157.859
C03282=1036.097,153.871,399.776,169.748,41.673,157.859
C03283=1036.104,154.119,399.754,169.751,41.673,157.859
C03284=1036.109,154.369,399.732,169.753,41.673,157.859
C03285=1036.115,154.617,399.709,169.756,41.672,157.860
C03286=1036.122,154.866,399.688,169.758,41.672,157.860
C03287=1036.127,155.115,399.665,169.761,41.671,157.860
C03288=1036.134,155.364,399.642,169.763,41.672,157.860
C03289=1036.140,155.613,399.621,169.766,41.671,157.860
C03290=1036.146,155.862,399.598,169.768,41.671,157.860
C03291=1036.152,156.111,399.576,169.771,41.671,157.860
C03292=1036.158,156.360,399.554,169.773,41.670,157.860
C03293=1036.165,156.645,399.529,169.776,41.670,157.860
C03294=1036.172,156.929,399.503,169.779,41.670,157.860
C03295=1036.179,157.215,399.478,169.783,41.669,157.860
C03296=1036.186,157.500,399.452,169.786,41.669,157.861
C03297=1036.192,157.749,399.429,169.789,41.669,157.861
C03298=1036.198,157.998,399.407,169.791,41.669,157.861
C03299=1036.203,158.247,399.384,169.794,41.668,157.861
C03300=1036.210,158.496,399.363,169.796,41.668,157.861
C03301=1036.216,158.744,399.341,169.799,41.668,157.861
C03302=1036.222,158.993,399.318,169.801,41.667,157.861
C03303=1036.228,159.243,399.296,169.804,41.668,157.861
C03304=1036.234,159.491,399.274,169.807,41.667,157.862
C03305=1036.241,159.741,399.250,169.809,41.667,157.862
C03306=1036.247,159.989,399.228,169.812,41.667,157.862
C03307=1036.253,160.239,399.206,169.814,41.666,157.862
C03308=1036.258,160.488,399.183,169.817,41.666,157.862
C03309=1036.265,160.736,399.160,169.820,41.666,157.862
C03310=1036.271,160.985,399.137,169.823,41.666,157.862
C03311=1036.276,161.234,399.114,169.825,41.666,157.862
C03312=1036.282,161.483,399.092,169.828,41.666,157.862
C03313=1036.289,161.732,399.069,169.830,41.665,157.863
C03314=1036.294,161.981,399.047,169.833,41.666,157.863
C03315=1036.300,162.230,399.024,169.836,41.665,157.863
C03316=1036.305,162.479,399.001,169.838,41.665,157.863
C03317=1036.312,162.727,398.979,169.841,41.665,157.863
C03318=1036.318,162.976,398.956,169.843,41.665,157.863
C03319=1036.323,163.225,398.933,169.847,41.665,157.864
C03320=1036.329,163.474,398.910,169.849,41.665,157.864
C03321=1036.335,163.723,398.887,169.852,41.665,157.864
C03322=1036.341,163.972,398.865,169.854,41.665,157.864
C03323=1036.347,164.221,398.842,169.857,41.664,157.864
C03324=1036.353,164.469,398.819,169.859,41.664,157.864
C03325=1036.358,164.718,398.796,169.862,41.664,157.864
C03326=1036.365,164.967,398.773,169.865,41.664,157.864
C03327=1036.371,165.216,398.750,169.867,41.664,157.864
C03328=1036.376,165.465,398.728,169.870,41.664,157.865
C03329=1036.382,165.714,398.705,169.872,41.664,157.865
C03330=1036.388,165.962,398.682,169.876,41.664,157.865
C03331=1036.395,166.212,398.659,169.879,41.664,157.865
C03332=1036.401,166.461,398.636,169.881,41.663,157.865
C03333=1036.406,166.710,398.613,169.884,41.663,157.865
C03334=1036.412,166.958,398.590,169.886,41.663,157.865
C03335=1036.418,167.207,398.567,169.889,41.663,157.866
C03336=1036.424,167.456,398.545,169.891,41.663,157.866
C03337=1036.430,167.705,398.522,169.894,41.663,157.866
C03338=1036.436,167.953,398.498,169.897,41.663,157.866
C03339=1036.442,168.203,398.475,169.899,41.663,157.866
C03340=1036.448,168.452,398.452,169.902,41.662,157.866
C03341=1036.455,168.700,398.430,169.906,41.663,157.866
C03342=1036.460,168.949,398.407,169.908,41.662,157.867
C03343=1036.466,169.198,398.384,169.911,41.662,157.867
C03344=1036.472,169.448,398.360,169.913,41.662,157.867
C03345=1036.478,169.696,398.337,169.916,41.662,157.867
C03346=1036.485,169.944,398.314,169.919,41.662,157.867
C03347=1036.491,170.193,398.291,169.921,41.662,157.867
C03348=1036.496,170.442,398.268,169.924,41.661,157.867
C03349=1036.503,170.692,398.245,169.927,41.662,157.868
C03350=1036.509,170.940,398.221,169.929,41.661,157.868
C03351=1036.514,171.189,398.199,169.933,41.662,157.868
C03352=1036.521,171.438,398.176,169.936,41.661,157.868
C03353=1036.527,171.686,398.153,169.938,41.661,157.868
C03354=1036.533,171.935,398.129,169.941,41.661,157.868
C03355=1036.539,172.184,398.106,169.944,41.661,157.868
C03356=1036.545,172.433,398.083,169.946,41.661,157.869
C03357=1036.553,172.718,398.057,169.949,41.661,157.869
C03358=1036.559,173.003,398.030,169.952,41.660,157.869
C03359=1036.566,173.287,398.004,169.955,41.660,157.869
C03360=1036.573,173.572,397.977,169.958,41.660,157.869
C03361=1036.579,173.820,397.954,169.962,41.660,157.869
C03362=1036.586,174.069,397.931,169.965,41.660,157.869
C03363=1036.591,174.318,397.908,169.967,41.660,157.870
C03364=1036.598,174.567,397.884,169.970,41.660,157.870
C03365=1036.603,174.815,397.861,169.973,41.659,157.870
C03366=1036.610,175.065,397.838,169.976,41.660,157.870
C03367=1036.616,175.313,397.815,169.978,41.659,157.870
C03368=1036.622,175.562,397.792,169.981,41.660,157.870
C03369=1036.629,175.811,397.768,169.985,41.659,157.870
C03370=1036.634,176.060,397.745,169.987,41.660,157.871
C03371=1036.640,176.309,397.722,169.990,41.659,157.871
C03372=1036.647,176.558,397.698,169.993,41.659,157.871
C03373=1036.653,176.807,397.675,169.996,41.659,157.871
C03374=1036.660,177.055,397.652,169.998,41.659,157.871
C03375=1036.666,177.304,397.629,170.001,41.659,157.871
C03376=1036.672,177.552,397.605,170.004,41.658,157.872
C03377=1036.678,177.802,397.582,170.006,41.659,157.872
C03378=1036.684,178.050,397.558,170.009,41.658,157.872
C03379=1036.690,178.299,397.535,170.013,41.658,157.872
C03380=1036.696,178.548,397.511,170.016,41.658,157.872
C03381=1036.702,178.797,397.488,170.018,41.658,157.872
C03382=1036.710,179.046,397.465,170.021,41.658,157.872
C03383=1036.715,179.295,397.442,170.024,41.658,157.873
C03384=1036.722,179.544,397.418,170.027,41.658,157.873
C03385=1036.728,179.793,397.395,170.030,41.658,157.873
C03386=1036.734,180.041,397.371,170.032,41.658,157.873
C03387=1036.740,180.290,397.348,170.036,41.658,157.873
C03388=1036.746,180.539,397.324,170.039,41.657,157.873
C03389=1036.753,180.788,397.300,170.042,41.657,157.874
C03390=1036.759,181.036,397.278,170.044,41.657,157.874
C03391=1036.766,181.285,397.254,170.047,41.657,157.874
C03392=1036.772,181.534,397.231,170.050,41.657,157.874
C03393=1036.778,181.783,397.207,170.053,41.657,157.874
C03394=1036.784,182.031,397.183,170.056,41.657,157.874
C03395=1036.791,182.281,397.160,170.058,41.657,157.874
C03396=1036.797,182.529,397.136,170.062,41.657,157.875
C03397=1036.803,182.778,397.112,170.065,41.657,157.875
C03398=1036.809,183.027,397.089,170.068,41.657,157.875
C03399=1036.816,183.276,397.066,170.071,41.657,157.875
C03400=1036.822,183.524,397.041,170.073,41.656,157.875
C03401=1036.828,183.773,397.017,170.076,41.657,157.875
C03402=1036.834,184.022,396.993,170.079,41.657,157.876
C03403=1036.840,184.270,396.970,170.082,41.657,157.876
C03404=1036.845,184.520,396.946,170.085,41.657,157.876
C03405=1036.851,184.768,396.922,170.088,41.657,157.876
C03406=1036.857,185.018,396.897,170.091,41.657,157.876
C03407=1036.863,185.266,396.874,170.093,41.658,157.877
C03408=1036.870,185.515,396.850,170.097,41.658,157.877
C03409=1036.875,185.764,396.825,170.100,41.657,157.877
C03410=1036.882,186.013,396.801,170.103,41.658,157.877
C03411=1036.887,186.261,396.777,170.105,41.658,157.877
C03412=1036.894,186.510,396.753,170.108,41.658,157.878
C03413=1036.899,186.759,396.729,170.111,41.659,157.878
C03414=1036.905,187.007,396.705,170.115,41.659,157.878
C03415=1036.911,187.256,396.681,170.117,41.658,157.878
C03416=1036.917,187.505,396.657,170.120,41.659,157.878
C03417=1036.923,187.754,396.632,170.123,41.659,157.879
C03418=1036.929,188.002,396.609,170.126,41.659,157.879
C03419=1036.935,188.251,396.584,170.129,41.659,157.879
C03420=1036.941,188.500,396.560,170.131,41.659,157.879
C03421=1036.948,188.784,396.532,170.136,41.659,157.879
C03422=1036.955,189.069,396.505,170.139,41.659,157.880
C03423=1036.962,189.352,396.477,170.142,41.660,157.880
C03424=1036.969,189.637,396.449,170.145,41.660,157.880
C03425=1036.975,189.885,396.425,170.149,41.660,157.880
C03426=1036.981,190.134,396.401,170.152,41.660,157.881
C03427=1036.987,190.383,396.377,170.155,41.661,157.881
C03428=1036.993,190.632,396.353,170.157,41.661,157.881
C03429=1036.999,190.881,396.328,170.160,41.661,157.881
C03430=1037.005,191.129,396.304,170.163,41.661,157.881
C03431=1037.011,191.378,396.279,170.167,41.661,157.882
C03432=1037.017,191.626,396.255,170.170,41.661,157.882
C03433=1037.023,191.875,396.231,170.173,41.661,157.882
C03434=1037.030,192.124,396.207,170.175,41.662,157.882
C03435=1037.036,192.372,396.182,170.178,41.662,157.883
C03436=1037.041,192.622,396.157,170.182,41.662,157.883
C03437=1037.047,192.870,396.133,170.185,41.662,157.883
C03438=1037.053,193.119,396.109,170.188,41.662,157.883
C03439=1037.060,193.368,396.084,170.191,41.662,157.883
C03440=1037.066,193.616,396.060,170.194,41.662,157.884
C03441=1037.072,193.865,396.036,170.197,41.663,157.884
C03442=1037.078,194.114,396.011,170.200,41.663,157.884
C03443=1037.085,194.362,395.987,170.203,41.663,157.884
C03444=1037.090,194.611,395.962,170.206,41.663,157.884
C03445=1037.097,194.860,395.938,170.209,41.664,157.885
C03446=1037.103,195.109,395.913,170.213,41.664,157.885
C03447=1037.109,195.357,395.889,170.216,41.664,157.885
C03448=1037.115,195.606,395.864,170.219,41.664,157.885
C03449=1037.122,195.855,395.840,170.221,41.664,157.885
C03450=1037.127,196.104,395.815,170.224,41.664,157.886
C03451=1037.134,196.352,395.791,170.228,41.664,157.886
C03452=1037.140,196.601,395.766,170.231,41.665,157.886
C03453=1037.147,196.850,395.742,170.234,41.665,157.886
C03454=1037.153,197.098,395.717,170.237,41.665,157.887
C03455=1037.158,197.347,395.692,170.240,41.665,157.887
C03456=1037.165,197.596,395.668,170.244,41.666,157.887
C03457=1037.171,197.845,395.643,170.247,41.666,157.887
C03458=1037.178,198.093,395.618,170.250,41.666,157.888
C03459=1037.183,198.342,395.594,170.253,41.666,157.888
C03460=1037.190,198.590,395.569,170.256,41.666,157.888
C03461=1037.196,198.840,395.545,170.259,41.667,157.888
C03462=1037.203,199.088,395.520,170.262,41.667,157.889
C03463=1037.209,199.337,395.495,170.265,41.667,157.889
C03464=1037.215,199.585,395.470,170.268,41.667,157.889
C03465=1037.221,199.834,395.446,170.272,41.668,157.889
C03466=1037.228,200.083,395.421,170.275,41.668,157.889
C03467=1037.234,200.332,395.397,170.278,41.668,157.890
C03468=1037.240,200.581,395.372,170.281,41.668,157.890
C03469=1037.247,200.829,395.347,170.284,41.669,157.890
C03470=1037.253,201.077,395.323,170.288,41.669,157.890
C03471=1037.259,201.326,395.297,170.291,41.669,157.891
C03472=1037.265,201.575,395.272,170.294,41.669,157.891
C03473=1037.271,201.824,395.247,170.297,41.669,157.891
C03474=1037.277,202.073,395.222,170.301,41.670,157.891
C03475=1037.283,202.321,395.197,170.304,41.671,157.892
C03476=1037.289,202.569,395.172,170.307,41.671,157.892
C03477=1037.295,202.819,395.147,170.310,41.671,157.892
C03478=1037.302,203.067,395.122,170.313,41.671,157.892
C03479=1037.308,203.316,395.097,170.317,41.672,157.893
C03480=1037.314,203.564,395.072,170.319,41.672,157.893
C03481=1037.321,203.813,395.046,170.322,41.673,157.893
C03482=1037.326,204.062,395.022,170.325,41.673,157.893
C03483=1037.332,204.310,394.997,170.329,41.674,157.894
C03484=1037.338,204.559,394.971,170.332,41.674,157.894
C03485=1037.364,205.610,394.865,170.639,41.778,157.934
C03486=1037.373,205.931,394.831,170.642,41.779,157.934
C03487=1037.382,206.253,394.797,170.645,41.781,157.935
C03488=1037.391,206.575,394.763,170.648,41.782,157.935
C03489=1037.400,206.897,394.728,170.651,41.784,157.936
C03490=1037.406,207.146,394.701,170.653,41.785,157.936
C03491=1037.413,207.394,394.675,170.655,41.786,157.937
C03492=1037.420,207.643,394.649,170.658,41.787,157.937
C03493=1037.427,207.891,394.622,170.660,41.788,157.938
C03494=1037.433,208.140,394.596,170.663,41.789,157.938
C03495=1037.440,208.388,394.569,170.665,41.790,157.938
C03496=1037.447,208.636,394.543,170.668,41.791,157.939
C03497=1037.453,208.886,394.516,170.670,41.792,157.939
C03498=1037.460,209.134,394.490,170.672,41.794,157.939
C03499=1037.467,209.382,394.463,170.674,41.795,157.940
C03500=1037.473,209.631,394.436,170.676,41.796,157.940
C03501=1037.480,209.880,394.410,170.679,41.797,157.940
C03502=1037.487,210.128,394.384,170.681,41.798,157.941
C03503=1037.493,210.377,394.357,170.684,41.799,157.941
C03504=1037.501,210.625,394.329,170.686,41.800,157.942
C03505=1037.507,210.873,394.303,170.688,41.801,157.942
C03506=1037.514,211.122,394.276,170.691,41.802,157.942
C03507=1037.521,211.371,394.250,170.693,41.804,157.943
C03508=1037.527,211.618,394.223,170.696,41.805,157.943
C03509=1037.534,211.867,394.196,170.698,41.806,157.944
C03510=1037.540,212.116,394.169,170.701,41.807,157.944
C03511=1037.547,212.364,394.143,170.703,41.808,157.944
C03512=1037.553,212.613,394.115,170.706,41.809,157.945
C03513=1037.561,212.861,394.089,170.708,41.810,157.945
C03514=1037.566,213.110,394.062,170.710,41.812,157.946
C03515=1037.574,213.358,394.035,170.712,41.813,157.946
C03516=1037.580,213.607,394.008,170.714,41.814,157.946
C03517=1037.587,213.854,393.981,170.717,41.815,157.947
C03518=1037.593,214.103,393.954,170.719,41.816,157.947
C03519=1037.600,214.352,393.928,170.722,41.817,157.947
C03520=1037.606,214.600,393.901,170.724,41.818,157.948
C03521=1037.614,214.849,393.874,170.727,41.820,157.948
C03522=1037.620,215.097,393.846,170.729,41.821,157.949
C03523=1037.627,215.346,393.819,170.731,41.822,157.949
C03524=1037.633,215.594,393.793,170.734,41.823,157.949
C03525=1037.640,215.843,393.766,170.736,41.824,157.950
C03526=1037.647,216.091,393.739,170.739,41.825,157.950
C03527=1037.654,216.340,393.712,170.741,41.826,157.950
C03528=1037.660,216.588,393.685,170.743,41.827,157.951
C03529=1037.667,216.836,393.658,170.746,41.829,157.951
C03530=1037.674,217.085,393.631,170.748,41.830,157.952
C03531=1037.681,217.334,393.604,170.751,41.831,157.952
C03532=1037.686,217.582,393.577,170.753,41.832,157.952
C03533=1037.694,217.830,393.550,170.756,41.833,157.953
C03534=1037.700,218.079,393.523,170.758,41.834,157.953
C03535=1037.708,218.327,393.496,170.761,41.835,157.954
C03536=1037.714,218.576,393.469,170.764,41.836,157.954
C03537=1037.721,218.824,393.442,170.767,41.838,157.954
C03538=1037.727,219.073,393.415,170.769,41.839,157.955
C03539=1037.735,219.321,393.388,170.771,41.840,157.955
C03540=1037.741,219.570,393.361,170.774,41.841,157.955
C03541=1037.748,219.818,393.333,170.776,41.842,157.956
C03542=1037.756,220.145,393.297,170.779,41.844,157.956
C03543=1037.766,220.473,393.261,170.782,41.845,157.957
C03544=1037.774,220.800,393.225,170.786,41.847,157.958
C03545=1037.783,221.128,393.189,170.789,41.848,157.958
C03546=1037.789,221.377,393.162,170.792,41.849,157.958
C03547=1037.795,221.625,393.135,170.795,41.851,157.959
C03548=1037.802,221.873,393.107,170.797,41.852,157.959
C03549=1037.809,222.122,393.079,170.799,41.853,157.960
C03550=1037.816,222.370,393.053,170.802,41.854,157.960
C03551=1037.823,222.619,393.025,170.804,41.855,157.960
C03552=1037.829,222.867,392.997,170.807,41.856,157.961
C03553=1037.835,223.115,392.970,170.809,41.858,157.961
C03554=1037.842,223.364,392.942,170.812,41.859,157.962
C03555=1037.848,223.613,392.915,170.814,41.860,157.962
C03556=1037.856,223.861,392.888,170.817,41.861,157.962
C03557=1037.862,224.109,392.860,170.819,41.862,157.963
C03558=1037.869,224.358,392.833,170.821,41.863,157.963
C03559=1037.876,224.606,392.805,170.824,41.865,157.964
C03560=1037.882,224.855,392.777,170.827,41.866,157.964
C03561=1037.888,225.103,392.751,170.830,41.867,157.964
C03562=1037.896,225.351,392.723,170.832,41.868,157.965
C03563=1037.902,225.599,392.696,170.835,41.869,157.965
C03564=1037.909,225.848,392.668,170.837,41.870,157.966
C03565=1037.916,226.096,392.640,170.840,41.872,157.966
C03566=1037.922,226.345,392.613,170.842,41.873,157.966
C03567=1037.929,226.593,392.585,170.845,41.874,157.967
C03568=1037.936,226.842,392.557,170.847,41.875,157.967
C03569=1037.943,227.090,392.530,170.851,41.876,157.968
C03570=1037.950,227.338,392.502,170.853,41.877,157.968
C03571=1037.956,227.587,392.475,170.855,41.879,157.969
C03572=1037.963,227.836,392.447,170.858,41.879,157.969
C03573=1037.970,228.084,392.420,170.860,41.880,157.969
C03574=1037.976,228.333,392.392,170.863,41.882,157.970
C03575=1037.983,228.581,392.364,170.865,41.883,157.970
C03576=1037.990,228.829,392.336,170.869,41.884,157.970
C03577=1037.996,229.077,392.308,170.871,41.885,157.971
C03578=1038.003,229.325,392.281,170.874,41.886,157.971
C03579=1038.009,229.573,392.253,170.876,41.888,157.972
C03580=1038.016,229.822,392.225,170.879,41.889,157.972
C03581=1038.023,230.070,392.198,170.881,41.890,157.973
C03582=1038.029,230.319,392.170,170.884,41.891,157.973
C03583=1038.035,230.568,392.142,170.886,41.892,157.973
C03584=1038.042,230.816,392.114,170.890,41.894,157.974
C03585=1038.049,231.064,392.085,170.892,41.895,157.974
C03586=1038.056,231.312,392.058,170.895,41.896,157.975
C03587=1038.062,231.561,392.030,170.897,41.897,157.975
C03588=1038.069,231.809,392.002,170.899,41.898,157.975
C03589=1038.076,232.058,391.974,170.902,41.900,157.976
C03590=1038.083,232.305,391.946,170.905,41.901,157.976
C03591=1038.089,232.554,391.918,170.908,41.902,157.977
C03592=1038.095,232.803,391.890,170.910,41.903,157.977
C03593=1038.102,233.051,391.862,170.913,41.905,157.978
C03594=1038.109,233.299,391.834,170.915,41.906,157.978
C03595=1038.115,233.548,391.805,170.918,41.907,157.979
C03596=1038.122,233.796,391.778,170.921,41.908,157.979
C03597=1038.128,234.044,391.750,170.924,41.910,157.979
C03598=1038.137,234.364,391.714,170.927,41.911,157.980
C03599=1038.146,234.685,391.677,170.931,41.912,157.980
C03600=1038.154,235.004,391.640,170.934,41.914,157.981
C03601=1038.163,235.325,391.605,170.937,41.915,157.981
C03602=1038.169,235.573,391.576,170.940,41.917,157.982
C03603=1038.176,235.821,391.548,170.943,41.918,157.982
C03604=1038.183,236.069,391.520,170.946,41.919,157.983
C03605=1038.189,236.318,391.492,170.948,41.920,157.983
C03606=1038.196,236.567,391.463,170.951,41.922,157.984
C03607=1038.203,236.815,391.435,170.954,41.923,157.984
C03608=1038.210,237.063,391.407,170.956,41.924,157.984
C03609=1038.217,237.311,391.379,170.959,41.925,157.985
C03610=1038.223,237.560,391.350,170.961,41.926,157.985
C03611=1038.230,237.808,391.322,170.964,41.928,157.986
C03612=1038.236,238.056,391.294,170.967,41.929,157.986
C03613=1038.243,238.304,391.266,170.970,41.930,157.987
C03614=1038.249,238.553,391.237,170.972,41.931,157.987
C03615=1038.257,238.801,391.209,170.975,41.933,157.988
C03616=1038.263,239.050,391.181,170.978,41.934,157.988
C03617=1038.270,239.298,391.152,170.981,41.935,157.988
C03618=1038.276,239.546,391.124,170.983,41.936,157.989
C03619=1038.283,239.794,391.096,170.987,41.937,157.989
C03620=1038.289,240.043,391.067,170.989,41.938,157.990
C03621=1038.297,240.291,391.039,170.992,41.940,157.990
C03622=1038.304,240.539,391.010,170.994,41.941,157.990
C03623=1038.310,240.788,390.982,170.998,41.942,157.991
C03624=1038.317,241.036,390.953,171.000,41.943,157.991
C03625=1038.323,241.284,390.924,171.003,41.945,157.992
C03626=1038.330,241.532,390.897,171.005,41.946,157.992
C03627=1038.337,241.781,390.867,171.009,41.947,157.993
C03628=1038.343,242.029,390.838,171.012,41.949,157.993
C03629=1038.350,242.278,390.810,171.014,41.950,157.994
C03630=1038.356,242.526,390.781,171.016,41.951,157.994
C03631=1038.363,242.774,390.753,171.020,41.952,157.994
C03632=1038.369,243.022,390.724,171.022,41.954,157.995
C03633=1038.376,243.271,390.696,171.025,41.955,157.995
C03634=1038.383,243.519,390.667,171.028,41.956,157.996
C03635=1038.389,243.767,390.638,171.031,41.958,157.996
C03636=1038.396,244.015,390.609,171.033,41.959,157.997
C03637=1038.402,244.263,390.580,171.037,41.960,157.997
C03638=1038.409,244.512,390.552,171.040,41.962,157.998
C03639=1038.416,244.760,390.523,171.042,41.963,157.998
C03640=1038.423,245.008,390.495,171.045,41.964,157.999
